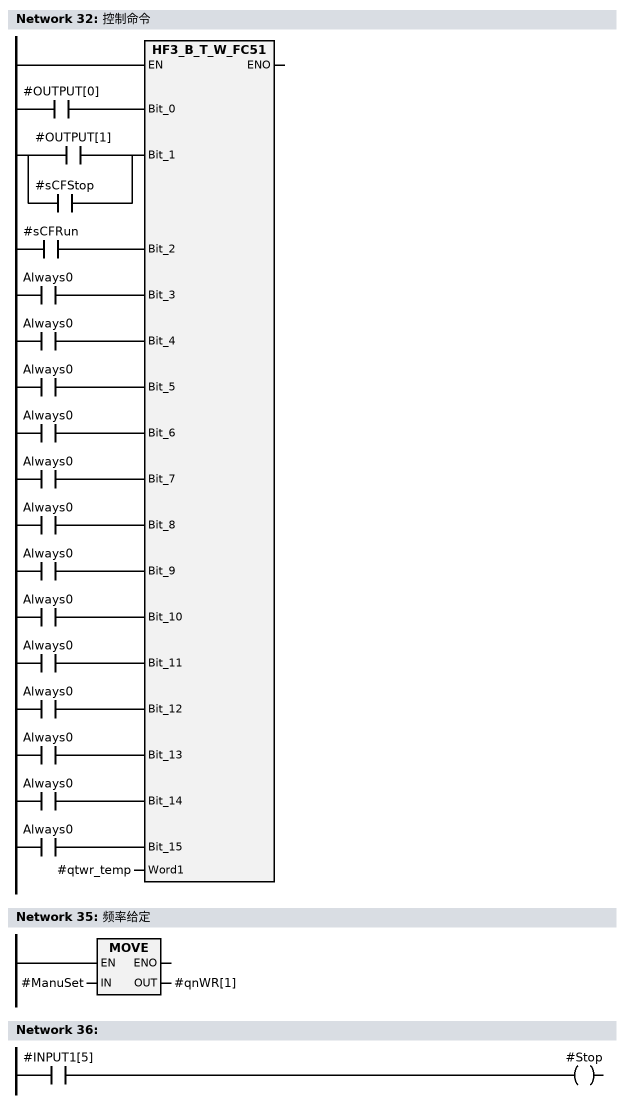
[picture p49: HF3_IMCC_TEF_FB2662 networks 32-36]
NETWORK
TITLE = 控制命令
      A     #OUTPUT[0];
      =     L 10.0;
      BLD   103;
      A(;
      O     #OUTPUT[1];
      O     #sCFStop;
      );
      =     L 10.1;
      BLD   103;
      A     #sCFRun;
      =     L 10.2;
      BLD   103;
      A     "Always0";
      =     L 10.3;
      BLD   103;
      A     "Always0";
      =     L 10.4;
      BLD   103;
      A     "Always0";
      =     L 10.5;
      BLD   103;
      A     "Always0";
      =     L 10.6;
      BLD   103;
      A     "Always0";
      =     L 10.7;
      BLD   103;
      A     "Always0";
      =     L 11.0;
      BLD   103;
      A     "Always0";
      =     L 11.1;
      BLD   103;
      A     "Always0";
      =     L 11.2;
      BLD   103;
      A     "Always0";
      =     L 11.3;
      BLD   103;
      A     "Always0";
      =     L 11.4;
      BLD   103;
      A     "Always0";
      =     L 11.5;
      BLD   103;
      A     "Always0";
      =     L 11.6;
      BLD   103;
      A     "Always0";
      =     L 11.7;
      BLD   103;
      CALL  "HF3_B_T_W_FC51" (
           Bit_0                    := L 10.0,
           Bit_1                    := L 10.1,
           Bit_2                    := L 10.2,
           Bit_3                    := L 10.3,
           Bit_4                    := L 10.4,
           Bit_5                    := L 10.5,
           Bit_6                    := L 10.6,
           Bit_7                    := L 10.7,
           Bit_8                    := L 11.0,
           Bit_9                    := L 11.1,
           Bit_10                   := L 11.2,
           Bit_11                   := L 11.3,
           Bit_12                   := L 11.4,
           Bit_13                   := L 11.5,
           Bit_14                   := L 11.6,
           Bit_15                   := L 11.7,
           Word1                    := #qtwr_temp);
      NOP   0;
NETWORK
TITLE = 参数传递
//控制命令输出
      CLR;
      L     #SCtrl;
      L     W#16#ABCD;
      <>I;
      JC    seiz;
      L     W#16#0;
      T     #qtwr_temp;
seiz: L     #qtwr_temp;
      T     #qnWR[0];
//tohmi输出
      L     #HMI_Adr;
      SLD   3;
      LAR1;
      OPN   DB [#DB_NO];
      L     #TOHMI_1;
      T     DBW [AR1,P#0.0];
      L     #TOHMI_2;
      T     DBW [AR1,P#2.0];
NETWORK
TITLE = 运行时间 故障次数
      A(;
      O     #INPUT1[3];
      O     #INPUT1[4];
      );
      =     L 10.0;
      BLD   103;
      A     #Flt;
      =     L 10.1;
      BLD   103;
      A     M 20.3;
      =     L 10.2;
      BLD   103;
      A     #SCtrl_Temp[12];
      =     L 10.4;
      BLD   103;
      A     #SCtrl_Temp[13];
      =     L 10.5;
      BLD   103;
      BLD   14;
      =     L 17.0;
      L     DINO;
      T     LW 15;
      CDB;
      OPN   DI [LW 15];
      TAR2  LD 11;
      A     L 10.0;
      =     DIX [AR2,P#136.0];
      A     L 10.1;
      =     DIX [AR2,P#136.1];
      A     L 10.2;
      =     DIX [AR2,P#136.2];
      A     L 10.4;
      =     DIX [AR2,P#136.4];
      A     L 10.5;
      =     DIX [AR2,P#136.5];
      +AR2  P#136.0;
      UC    "HF3_RunFaultSum";
      LAR2  LD 11;
      L     DID [AR2,P#138.0];
      T     DBD [AR2,P#58.0];
      L     DIW [AR2,P#142.0];
      T     DBW [AR2,P#64.0];
      L     DIW [AR2,P#144.0];
      T     DBW [AR2,P#62.0];
      CDB;
      BLD   15;
      NOP   0;
NETWORK
TITLE = 频率给定
      L     #ManuSet;
      T     #qnWR[1];
      NOP   0;
NETWORK
TITLE =
      A     #INPUT1[5];
      =     #Stop;
END_FUNCTION_BLOCK

FUNCTION_BLOCK "HF3_IMCC_KT_FB2671"	// FB 2671
VERSION : 0.1
VAR
  PT : TIME  := T#45S;
  KT_B1 : FB 2672;
END_VAR
BEGIN
NETWORK
TITLE =
// (network holds code this reader does not know; not shown)
END_FUNCTION_BLOCK

FUNCTION_BLOCK "HF3_IMCC_KT_FB2672"	// FB 2672
VERSION : 0.1
VAR_INPUT
  Main : BOOL ;	//1为大端 0为小端
  IN_RD : ARRAY  [0 .. 10 ] OF WORD ;
  HMI_Adr : INT ;
  SCtrl : WORD ;	//0单控1模控2启动3停止
  MCtrl : ARRAY  [0 .. 3 ] OF //模式控制
  BOOL ;
  Mode : ARRAY  [0 .. 15 ] OF //模式执行状态
  BOOL ;
  Open : BOOL ;	//风阀开连锁
  PT : TIME ;	//执行时间
  ALL : ARRAY  [0 .. 15 ] OF //单系统命令
  BOOL ;
  H_P_All_Ctrl : WORD ;	//全局命令
  FireAlarm : BOOL ;	//火灾报警
  BlockAlarm : BOOL ;	//阻塞报警
  ManuSet : INT ;	//手动频率给定
END_VAR
VAR_OUTPUT
  qnWR : ARRAY  [0 .. 1 ] OF WORD ;
  RT : REAL ;
  SumFlt : INT ;
  SumRun : INT ;
  refuse : BOOL ;
  Stop : BOOL ;	//风机控制
END_VAR
VAR
  IN_RD1 : WORD ;
  qtWR_1 : WORD ;
  TOHMI_1 : WORD ;
  TOHMI_2 : WORD ;
  qtwr_temp : WORD ;
  SFlag : BOOL ;	//单控标志
  McFlag : BOOL ;	//检修牌
  QTout : BOOL ;	//输出超时
  Flt : BOOL ;	//设备综合故障
  SingTout : BOOL ;	//单控超时
  Timeout : BOOL ;	//设备动作超时
  PID_EN : BOOL ;	//pid使能
  Fault : BOOL ;	//故障
  sCFRun : BOOL ;	//火灾启动
  sCFStop : BOOL ;	//火灾停止
  INPUT1 : ARRAY  [0 .. 15 ] OF //设备状态字
  BOOL ;
  OUTPUT : ARRAY  [0 .. 15 ] OF //输出状态字
  BOOL ;
  Ctrl : ARRAY  [0 .. 15 ] OF BOOL ;
  SCtrl_Temp : ARRAY  [0 .. 15 ] OF //HMI命令
  BOOL ;
  Latch : ARRAY  [0 .. 7 ] OF BOOL ;
  temp : ARRAY  [0 .. 1 ] OF BOOL ;
  h_P_all_temp : ARRAY  [0 .. 15 ] OF BOOL ;
  ton1 : SFB 4;
  ton2 : SFB 4;
  RunFaultSum : FB 2006;
END_VAR
VAR_TEMP
  AR2_Value : DWORD ;
  DI_NO : INT ;
  Data_Len : INT ;
  DB_NO : INT ;
END_VAR
BEGIN
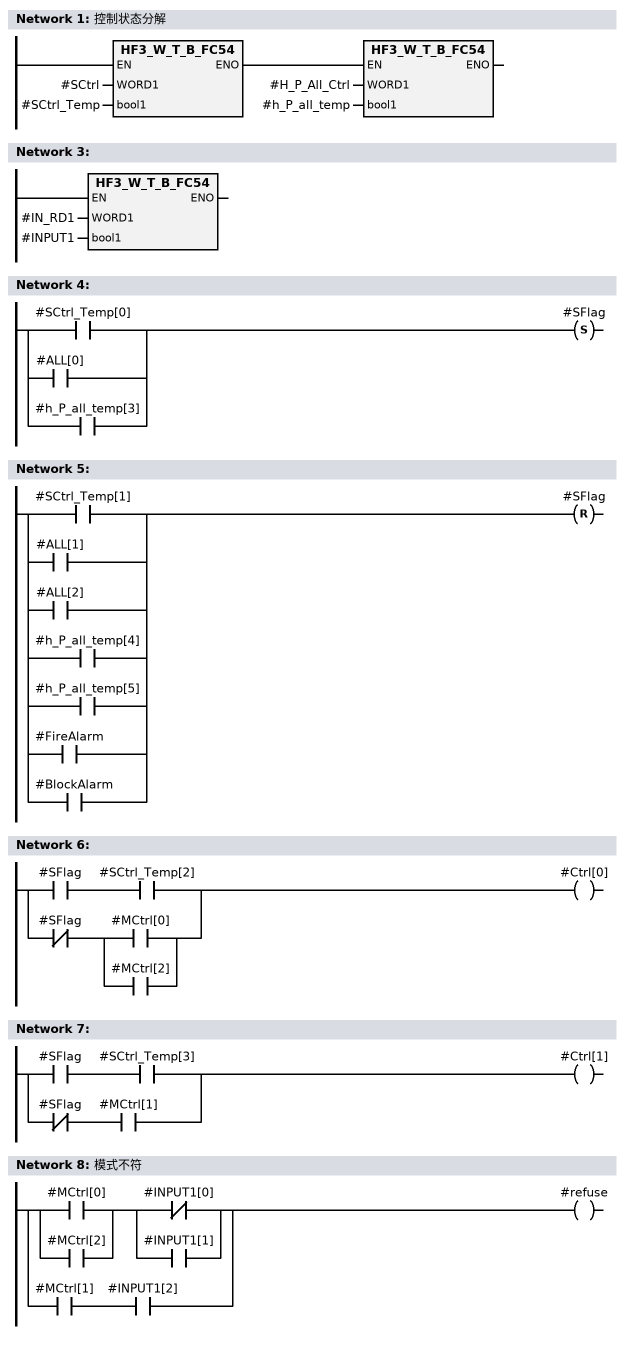
NETWORK
TITLE = 控制状态分解
      A(;
      CALL  "HF3_W_T_B_FC54" (
           WORD1                    := #SCtrl,
           bool1                    := #SCtrl_Temp);
      A     BR;
      );
      JNB   _001;
      CALL  "HF3_W_T_B_FC54" (
           WORD1                    := #H_P_All_Ctrl,
           bool1                    := #h_P_all_temp);
_001: NOP   0;
NETWORK
TITLE =
      TAR2;
      T     #AR2_Value;
      L     6002;
      T     #DB_NO;
      A     #Main;	//此端是否为大端
      JC    big;
      L     6004;
      T     #DB_NO;
big:  L     DINO;	//存储背景数据块号
      T     #DI_NO;
      OPN   DB [#DB_NO];	//打开
      L     #HMI_Adr;
      SLD   3;
      LAR1;
// *********************事故风机中DI状态读取**********************
      L     #IN_RD[0];	//第一个字中包含数字量信息
      T     #IN_RD1;
//初始化AR2寄存器用于AI量传递
      TAR2;
      AD    DW#16#FFFFFF;
      L     P##IN_RD;
      +D;
      OD    DW#16#85000000;
      LAR2;
//*********************事故风机中AI状态读取**********************
//读取模拟量输入
      L     13;
ilop: T     #Data_Len;
      L     W [AR2,P#2.0];	//智能低压点表新更新，第二个字开始为模拟量
      T     DBW [AR1,P#4.0];
      +AR1  P#2.0;
      +AR2  P#2.0;
      L     #Data_Len;
      LOOP  ilop;
//恢复AR2 DI寄存器
      L     #AR2_Value;
      LAR2;
//     OPN   DI [#DI_NO]
NETWORK
TITLE =
      CALL  "HF3_W_T_B_FC54" (
           WORD1                    := #IN_RD1,
           bool1                    := #INPUT1);
      NOP   0;
NETWORK
TITLE =
      O     #SCtrl_Temp[0];
      O     #ALL[0];
      O     #h_P_all_temp[3];
      S     #SFlag;
NETWORK
TITLE =
      O     #SCtrl_Temp[1];
      O     #ALL[1];
      O     #ALL[2];
      O     #h_P_all_temp[4];
      O     #h_P_all_temp[5];
      O     #FireAlarm;
      O     #BlockAlarm;
      R     #SFlag;
NETWORK
TITLE =
      A     #SFlag;
      A     #SCtrl_Temp[2];
      O;
      AN    #SFlag;
      A(;
      O     #MCtrl[0];
      O     #MCtrl[2];
      );
      =     #Ctrl[0];
NETWORK
TITLE =
      A     #SFlag;
      A     #SCtrl_Temp[3];
      O;
      AN    #SFlag;
      A     #MCtrl[1];
      =     #Ctrl[1];
NETWORK
TITLE = 模式不符
      A(;
      O     #MCtrl[0];
      O     #MCtrl[2];
      );
      A(;
      ON    #INPUT1[0];
      O     #INPUT1[1];
      );
      O;
      A     #MCtrl[1];
      A     #INPUT1[2];
      =     #refuse;
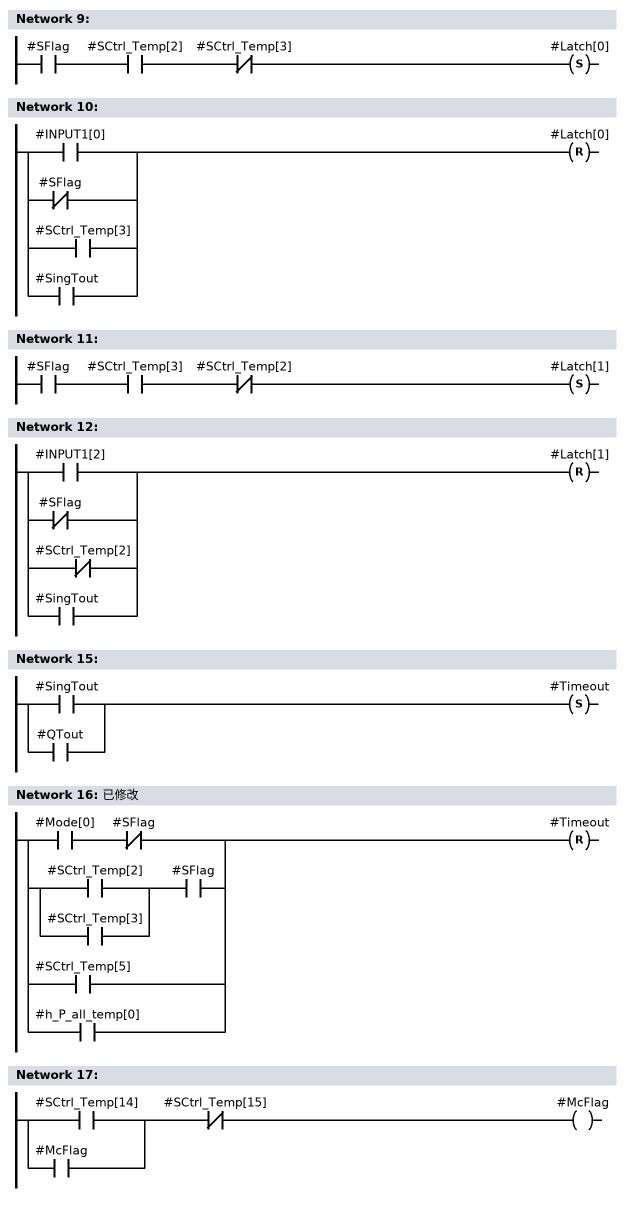
NETWORK
TITLE =
      A     #SFlag;
      A     #SCtrl_Temp[2];
      AN    #SCtrl_Temp[3];
      S     #Latch[0];
NETWORK
TITLE =
      O     #INPUT1[0];
      ON    #SFlag;
      O     #SCtrl_Temp[3];
      O     #SingTout;
      R     #Latch[0];
NETWORK
TITLE =
      A     #SFlag;
      A     #SCtrl_Temp[3];
      AN    #SCtrl_Temp[2];
      S     #Latch[1];
NETWORK
TITLE =
      O     #INPUT1[2];
      ON    #SFlag;
      ON    #SCtrl_Temp[2];
      O     #SingTout;
      R     #Latch[1];
NETWORK
TITLE =
      A(;
      O     #Latch[0];
      O     #Latch[1];
      );
      =     L 10.0;
      BLD   103;
      BLD   16;
      =     L 17.0;
      L     DINO;
      T     LW 15;
      CDB;
      OPN   DI [LW 15];
      TAR2  LD 11;
      A     L 10.0;
      =     DIX [AR2,P#86.0];
      L     DBD [AR2,P#34.0];
      T     DID [AR2,P#88.0];
      +AR2  P#86.0;
      UC    "TON";
      LAR2  LD 11;
      A     DIX [AR2,P#92.0];
      =     DBX [AR2,P#70.4];
      CDB;
      BLD   17;
      NOP   0;
NETWORK
TITLE =
      A(;
      O     #OUTPUT[0];
      O     #OUTPUT[1];
      );
      =     L 10.0;
      BLD   103;
      BLD   16;
      =     L 17.0;
      L     DINO;
      T     LW 15;
      CDB;
      OPN   DI [LW 15];
      TAR2  LD 11;
      A     L 10.0;
      =     DIX [AR2,P#108.0];
      L     DBD [AR2,P#34.0];
      T     DID [AR2,P#110.0];
      +AR2  P#108.0;
      UC    "TON";
      LAR2  LD 11;
      A     DIX [AR2,P#114.0];
      =     DBX [AR2,P#70.2];
      CDB;
      BLD   17;
      NOP   0;
NETWORK
TITLE =
      O     #SingTout;
      O     #QTout;
      S     #Timeout;
NETWORK
TITLE = 已修改
      A     #Mode[0];
      AN    #SFlag;
      O;
      A(;
      O     #SCtrl_Temp[2];
      O     #SCtrl_Temp[3];
      );
      A     #SFlag;
      O     #SCtrl_Temp[5];
      O     #h_P_all_temp[0];
      R     #Timeout;
NETWORK
TITLE =
      A(;
      O     #SCtrl_Temp[14];
      O     #McFlag;
      );
      AN    #SCtrl_Temp[15];
      =     #McFlag;
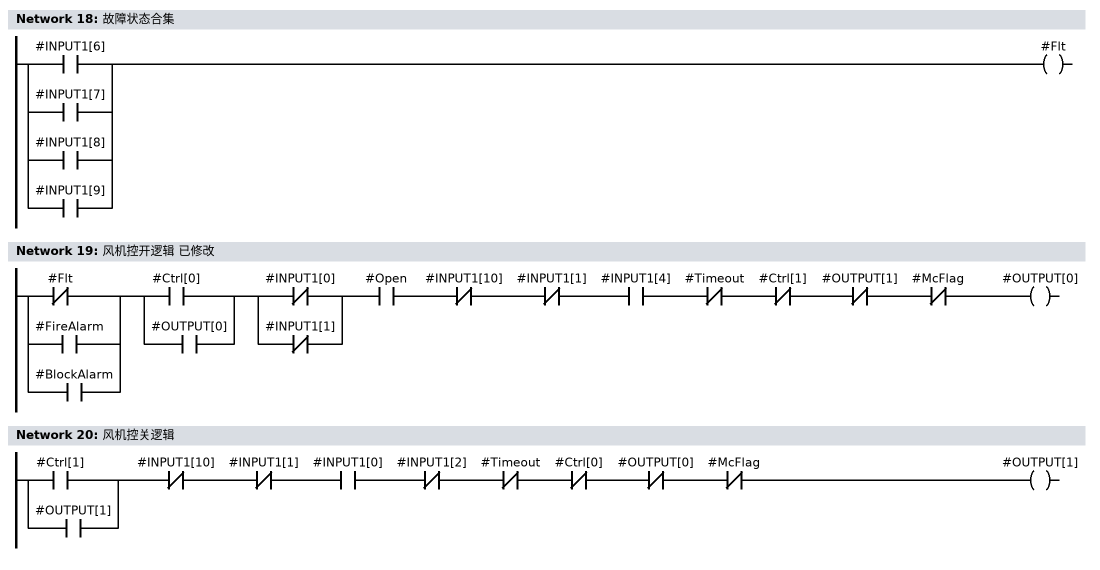
NETWORK
TITLE = 故障状态合集
      O     #INPUT1[6];
      O     #INPUT1[7];
      O     #INPUT1[8];
      O     #INPUT1[9];
      =     #Flt;
NETWORK
TITLE = 风机控开逻辑 已修改
      A(;
      ON    #Flt;
      O     #FireAlarm;
      O     #BlockAlarm;
      );
      A(;
      O     #Ctrl[0];
      O     #OUTPUT[0];
      );
      A(;
      ON    #INPUT1[0];
      ON    #INPUT1[1];
      );
      A     #Open;
      AN    #INPUT1[10];
      AN    #INPUT1[1];
      A     #INPUT1[4];
      AN    #Timeout;
      AN    #Ctrl[1];
      AN    #OUTPUT[1];
      AN    #McFlag;
      =     #OUTPUT[0];
NETWORK
TITLE = 风机控关逻辑
      A(;
      O     #Ctrl[1];
      O     #OUTPUT[1];
      );
      AN    #INPUT1[10];
      AN    #INPUT1[1];
      A     #INPUT1[0];
      AN    #INPUT1[2];
      AN    #Timeout;
      AN    #Ctrl[0];
      AN    #OUTPUT[0];
      AN    #McFlag;
      =     #OUTPUT[1];
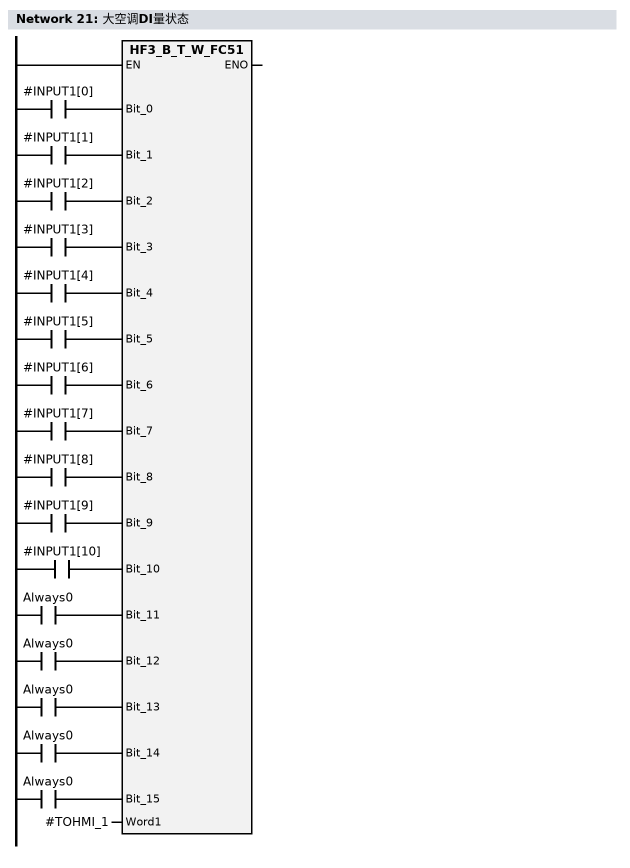
NETWORK
TITLE = 大空调DI量状态
      A     #INPUT1[0];
      =     L 10.0;
      BLD   103;
      A     #INPUT1[1];
      =     L 10.1;
      BLD   103;
      A     #INPUT1[2];
      =     L 10.2;
      BLD   103;
      A     #INPUT1[3];
      =     L 10.3;
      BLD   103;
      A     #INPUT1[4];
      =     L 10.4;
      BLD   103;
      A     #INPUT1[5];
      =     L 10.5;
      BLD   103;
      A     #INPUT1[6];
      =     L 10.6;
      BLD   103;
      A     #INPUT1[7];
      =     L 10.7;
      BLD   103;
      A     #INPUT1[8];
      =     L 11.0;
      BLD   103;
      A     #INPUT1[9];
      =     L 11.1;
      BLD   103;
      A     #INPUT1[10];
      =     L 11.2;
      BLD   103;
      A     "Always0";
      =     L 11.3;
      BLD   103;
      A     "Always0";
      =     L 11.4;
      BLD   103;
      A     "Always0";
      =     L 11.5;
      BLD   103;
      A     "Always0";
      =     L 11.6;
      BLD   103;
      A     "Always0";
      =     L 11.7;
      BLD   103;
      CALL  "HF3_B_T_W_FC51" (
           Bit_0                    := L 10.0,
           Bit_1                    := L 10.1,
           Bit_2                    := L 10.2,
           Bit_3                    := L 10.3,
           Bit_4                    := L 10.4,
           Bit_5                    := L 10.5,
           Bit_6                    := L 10.6,
           Bit_7                    := L 10.7,
           Bit_8                    := L 11.0,
           Bit_9                    := L 11.1,
           Bit_10                   := L 11.2,
           Bit_11                   := L 11.3,
           Bit_12                   := L 11.4,
           Bit_13                   := L 11.5,
           Bit_14                   := L 11.6,
           Bit_15                   := L 11.7,
           Word1                    := #TOHMI_1);
      NOP   0;
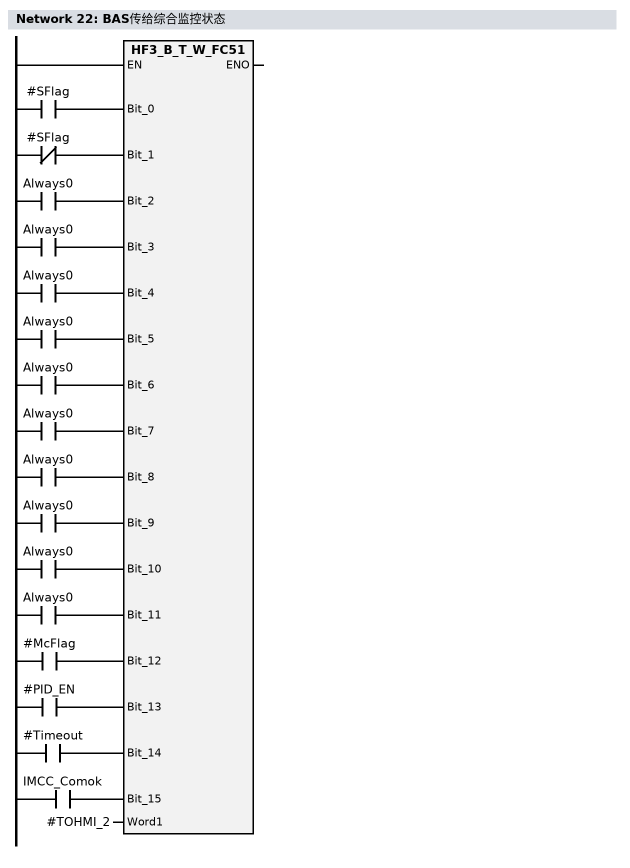
NETWORK
TITLE = BAS传给综合监控状态
//单模控、据动报警、检修牌、通讯状态
      A     #SFlag;
      =     L 10.0;
      BLD   103;
      AN    #SFlag;
      =     L 10.1;
      BLD   103;
      A     "Always0";
      =     L 10.2;
      BLD   103;
      A     "Always0";
      =     L 10.3;
      BLD   103;
      A     "Always0";
      =     L 10.4;
      BLD   103;
      A     "Always0";
      =     L 10.5;
      BLD   103;
      A     "Always0";
      =     L 10.6;
      BLD   103;
      A     "Always0";
      =     L 10.7;
      BLD   103;
      A     "Always0";
      =     L 11.0;
      BLD   103;
      A     "Always0";
      =     L 11.1;
      BLD   103;
      A     "Always0";
      =     L 11.2;
      BLD   103;
      A     "Always0";
      =     L 11.3;
      BLD   103;
      A     #McFlag;
      =     L 11.4;
      BLD   103;
      A     #PID_EN;
      =     L 11.5;
      BLD   103;
      A     #Timeout;
      =     L 11.6;
      BLD   103;
      A     "IMCC_Comok";
      =     L 11.7;
      BLD   103;
      CALL  "HF3_B_T_W_FC51" (
           Bit_0                    := L 10.0,
           Bit_1                    := L 10.1,
           Bit_2                    := L 10.2,
           Bit_3                    := L 10.3,
           Bit_4                    := L 10.4,
           Bit_5                    := L 10.5,
           Bit_6                    := L 10.6,
           Bit_7                    := L 10.7,
           Bit_8                    := L 11.0,
           Bit_9                    := L 11.1,
           Bit_10                   := L 11.2,
           Bit_11                   := L 11.3,
           Bit_12                   := L 11.4,
           Bit_13                   := L 11.5,
           Bit_14                   := L 11.6,
           Bit_15                   := L 11.7,
           Word1                    := #TOHMI_2);
      NOP   0;
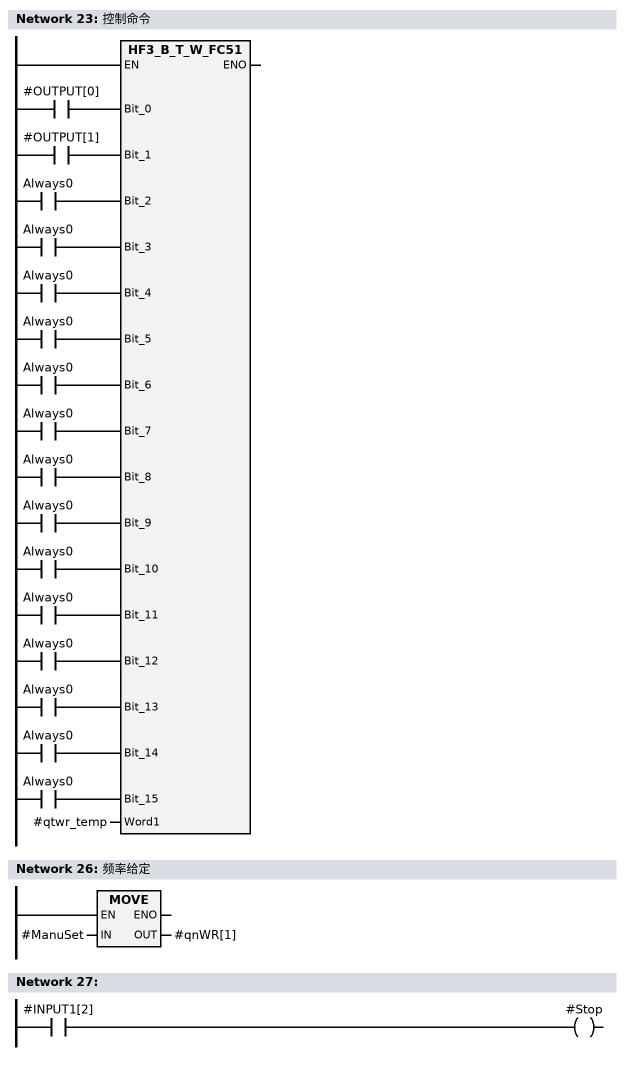
NETWORK
TITLE = 控制命令
      A     #OUTPUT[0];
      =     L 10.0;
      BLD   103;
      A     #OUTPUT[1];
      =     L 10.1;
      BLD   103;
      A     "Always0";
      =     L 10.2;
      BLD   103;
      A     "Always0";
      =     L 10.3;
      BLD   103;
      A     "Always0";
      =     L 10.4;
      BLD   103;
      A     "Always0";
      =     L 10.5;
      BLD   103;
      A     "Always0";
      =     L 10.6;
      BLD   103;
      A     "Always0";
      =     L 10.7;
      BLD   103;
      A     "Always0";
      =     L 11.0;
      BLD   103;
      A     "Always0";
      =     L 11.1;
      BLD   103;
      A     "Always0";
      =     L 11.2;
      BLD   103;
      A     "Always0";
      =     L 11.3;
      BLD   103;
      A     "Always0";
      =     L 11.4;
      BLD   103;
      A     "Always0";
      =     L 11.5;
      BLD   103;
      A     "Always0";
      =     L 11.6;
      BLD   103;
      A     "Always0";
      =     L 11.7;
      BLD   103;
      CALL  "HF3_B_T_W_FC51" (
           Bit_0                    := L 10.0,
           Bit_1                    := L 10.1,
           Bit_2                    := L 10.2,
           Bit_3                    := L 10.3,
           Bit_4                    := L 10.4,
           Bit_5                    := L 10.5,
           Bit_6                    := L 10.6,
           Bit_7                    := L 10.7,
           Bit_8                    := L 11.0,
           Bit_9                    := L 11.1,
           Bit_10                   := L 11.2,
           Bit_11                   := L 11.3,
           Bit_12                   := L 11.4,
           Bit_13                   := L 11.5,
           Bit_14                   := L 11.6,
           Bit_15                   := L 11.7,
           Word1                    := #qtwr_temp);
      NOP   0;
NETWORK
TITLE = 参数传递
//控制命令输出
      CLR;
      L     #SCtrl;
      L     W#16#ABCD;
      <>I;
      JC    seiz;
      L     W#16#0;
      T     #qtwr_temp;
seiz: L     #qtwr_temp;
      T     #qnWR[0];	//大空调开关控制字
//tohmi输出
      L     #HMI_Adr;
      SLD   3;
      LAR1;
      OPN   DB [#DB_NO];
      L     #TOHMI_1;
      T     DBW [AR1,P#0.0];
      L     #TOHMI_2;
      T     DBW [AR1,P#2.0];
NETWORK
TITLE =
      A(;
      O     #INPUT1[0];
      O     #INPUT1[1];
      );
      =     L 10.0;
      BLD   103;
      A     #Flt;
      =     L 10.1;
      BLD   103;
      A     M 20.5;
      =     L 10.2;
      BLD   103;
      A     #SCtrl_Temp[12];
      =     L 10.4;
      BLD   103;
      A     #SCtrl_Temp[13];
      =     L 10.5;
      BLD   103;
      BLD   14;
      =     L 17.0;
      L     DINO;
      T     LW 15;
      CDB;
      OPN   DI [LW 15];
      TAR2  LD 11;
      A     L 10.0;
      =     DIX [AR2,P#130.0];
      A     L 10.1;
      =     DIX [AR2,P#130.1];
      A     L 10.2;
      =     DIX [AR2,P#130.2];
      A     L 10.4;
      =     DIX [AR2,P#130.4];
      A     L 10.5;
      =     DIX [AR2,P#130.5];
      +AR2  P#130.0;
      UC    "HF3_RunFaultSum";
      LAR2  LD 11;
      L     DID [AR2,P#132.0];
      T     DBD [AR2,P#50.0];
      L     DIW [AR2,P#136.0];
      T     DBW [AR2,P#56.0];
      L     DIW [AR2,P#138.0];
      T     DBW [AR2,P#54.0];
      CDB;
      BLD   15;
      NOP   0;
NETWORK
TITLE = 频率给定
      L     #ManuSet;
      T     #qnWR[1];
      NOP   0;
NETWORK
TITLE =
      A     #INPUT1[2];
      =     #Stop;
END_FUNCTION_BLOCK

FUNCTION_BLOCK "HF3_IMCC_HPF_FB2681"	// FB 2681
VERSION : 0.1
VAR
  PT : TIME  := T#45S;
  HPF_A1 : FB 2682;
END_VAR
BEGIN
NETWORK
TITLE =
// (network holds code this reader does not know; not shown)
END_FUNCTION_BLOCK

FUNCTION_BLOCK "HF4_IMCC_HPF_FB2682"	// FB 2682
VERSION : 0.1
VAR_INPUT
  Main : BOOL ;
  IN_RD : ARRAY  [0 .. 7 ] OF WORD ;
  HMI_Adr : INT ;
  SCtrl : WORD ;	//01-单模23-启停
  MCtrl : ARRAY  [0 .. 3 ] OF //012-启动停止工频
  BOOL ;
  Mode : ARRAY  [0 .. 15 ] OF //012-开始结束时间表
  BOOL ;
  Open : BOOL ;	//连锁风阀开
  PT : TIME ;	//延迟时间
  ALL : ARRAY  [0 .. 15 ] OF //012-单控模控时间表
  BOOL ;
  H_P_All_Ctrl : WORD ;
  FireAlarm : BOOL ;	//火灾信号
  BlockAlarm : BOOL ;	//阻塞信号
  ManuSet : INT ;	//手动频率设定
END_VAR
VAR_OUTPUT
  qnWR : ARRAY  [0 .. 1 ] OF //0-频率1-启停
  WORD ;
  RT : REAL ;	//运行时间
  SumFlt : INT ;	//故障次数
  SumRun : INT ;	//运行次数
  Refuse : BOOL ;	//模式不符
  Stop : BOOL ;	//风机控制
END_VAR
VAR
  IN_RD1 : WORD ;
  qtWR : WORD ;
  TOHMI_1 : WORD ;
  TOHMI_2 : WORD ;
  qtwr_temp : WORD ;
  INPUT1 : ARRAY  [0 .. 15 ] OF BOOL ;
  OUTPUT : ARRAY  [0 .. 15 ] OF //01-启停
  BOOL ;
  Ctrl : ARRAY  [0 .. 15 ] OF //01-启停
  BOOL ;
  SCtrl_Temp : ARRAY  [0 .. 15 ] OF //01-单模23-启停
  BOOL ;
  H_P_All_Ctrl_Temp : ARRAY  [0 .. 15 ] OF BOOL ;
  Latch : ARRAY  [0 .. 7 ] OF //启停锁定
  BOOL ;
  McFlag : BOOL ;	//检修牌
  SFlag : BOOL ;	//单控标志
  SingTout : BOOL ;	//控制命令超时
  QTout : BOOL ;	//控制超时
  Timeout : BOOL ;	//超时
  Flt : BOOL ;	//设备综合故障
  PID_EN : BOOL ;	//PID使能
  Fault : BOOL ;
  TON1 : SFB 4;
  TON2 : SFB 4;
  RunFaultSum : FB 2006;
END_VAR
VAR_TEMP
  AR2_Value : DWORD ;
  DI_NO : INT ;
  Data_Len : INT ;
  DB_NO : INT ;
END_VAR
BEGIN
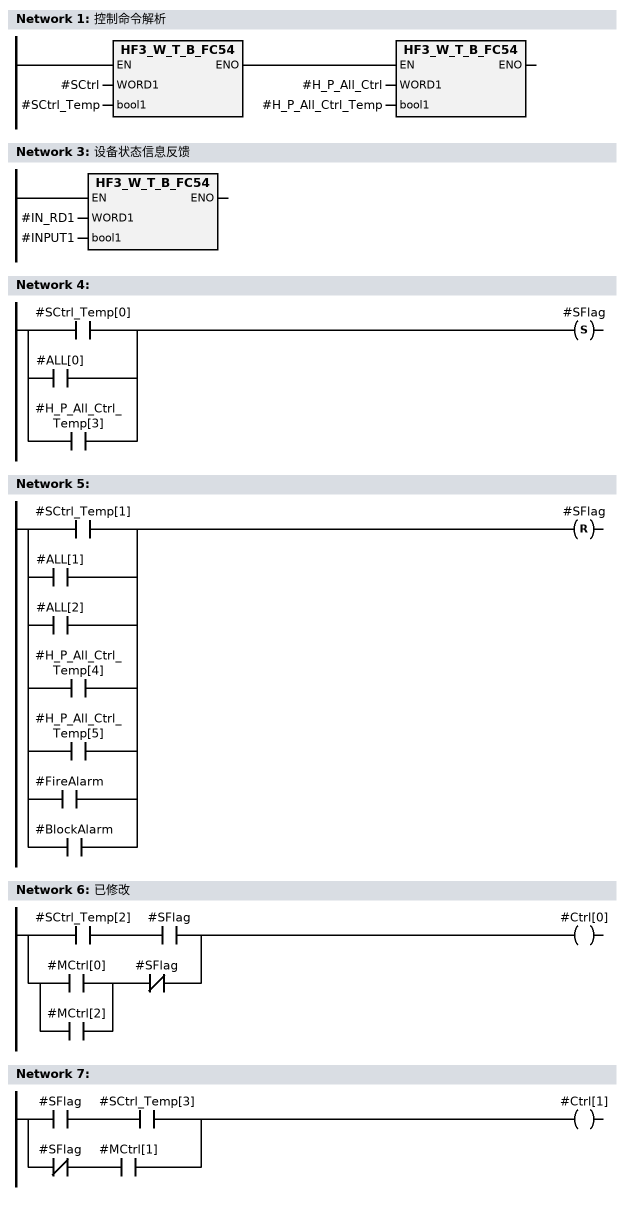
NETWORK
TITLE = 控制命令解析
      A(;
      CALL  "HF3_W_T_B_FC54" (
           WORD1                    := #SCtrl,
           bool1                    := #SCtrl_Temp);
      A     BR;
      );
      JNB   _001;
      CALL  "HF3_W_T_B_FC54" (
           WORD1                    := #H_P_All_Ctrl,
           bool1                    := #H_P_All_Ctrl_Temp);
_001: NOP   0;
NETWORK
TITLE = 状态信息读取
//第1个字BIT 0BAS
//第1个字BIT 1就地
//第1个字BIT 2变频/工频开关位置
//第1个字BIT 3变频运行状态
//第1个字BIT 4工频运行状态
//第1个字BIT 5变频器故障
//第1个字BIT 6变频器过载
//第1个字BIT 7电动机缺相
//
//
//第2个字频率反馈
//第3个字电动机电流A
//第4个字电动机电流B
//第5个字电动机电流C
//第6个字电动机电压A
//第7个字电动机电压B
//第8个字电动机电压C
//
      TAR2;
      T     #AR2_Value;
      L     6002;
      T     #DB_NO;
      A     #Main;	//此端是否为大端
      JC    big;
      L     6004;
      T     #DB_NO;
big:  L     DINO;	//存储背景数据块号
      T     #DI_NO;
      OPN   DB [#DB_NO];	//打开
      L     #HMI_Adr;
      SLD   3;
      LAR1;
// *********************事故风机中DI状态读取**********************
      L     #IN_RD[0];	//第一个字中包含数字量信息
      T     #IN_RD1;
//初始化AR2寄存器用于AI量传递
      TAR2;
      AD    DW#16#FFFFFF;
      L     P##IN_RD;
      +D;
      OD    DW#16#85000000;
      LAR2;
//*********************事故风机中AI状态读取**********************
//读取模拟量输入
      L     7;
ilop: T     #Data_Len;
      L     W [AR2,P#2.0];	//智能低压点表新更新，第二个字开始为模拟量
      T     DBW [AR1,P#4.0];
      +AR1  P#2.0;
      +AR2  P#2.0;
      L     #Data_Len;
      LOOP  ilop;
//恢复AR2 DI寄存器
      L     #AR2_Value;
      LAR2;
//     OPN   DI [#DI_NO]
NETWORK
TITLE = 设备状态信息反馈
      CALL  "HF3_W_T_B_FC54" (
           WORD1                    := #IN_RD1,
           bool1                    := #INPUT1);
      NOP   0;
NETWORK
TITLE =
      O     #SCtrl_Temp[0];
      O     #ALL[0];
      O     #H_P_All_Ctrl_Temp[3];
      S     #SFlag;
NETWORK
TITLE =
      O     #SCtrl_Temp[1];
      O     #ALL[1];
      O     #ALL[2];
      O     #H_P_All_Ctrl_Temp[4];
      O     #H_P_All_Ctrl_Temp[5];
      O     #FireAlarm;
      O     #BlockAlarm;
      R     #SFlag;
NETWORK
TITLE = 已修改
      A     #SCtrl_Temp[2];
      A     #SFlag;
      O;
      A(;
      O     #MCtrl[0];
      O     #MCtrl[2];
      );
      AN    #SFlag;
      =     #Ctrl[0];
NETWORK
TITLE =
      A     #SFlag;
      A     #SCtrl_Temp[3];
      O;
      AN    #SFlag;
      A     #MCtrl[1];
      =     #Ctrl[1];
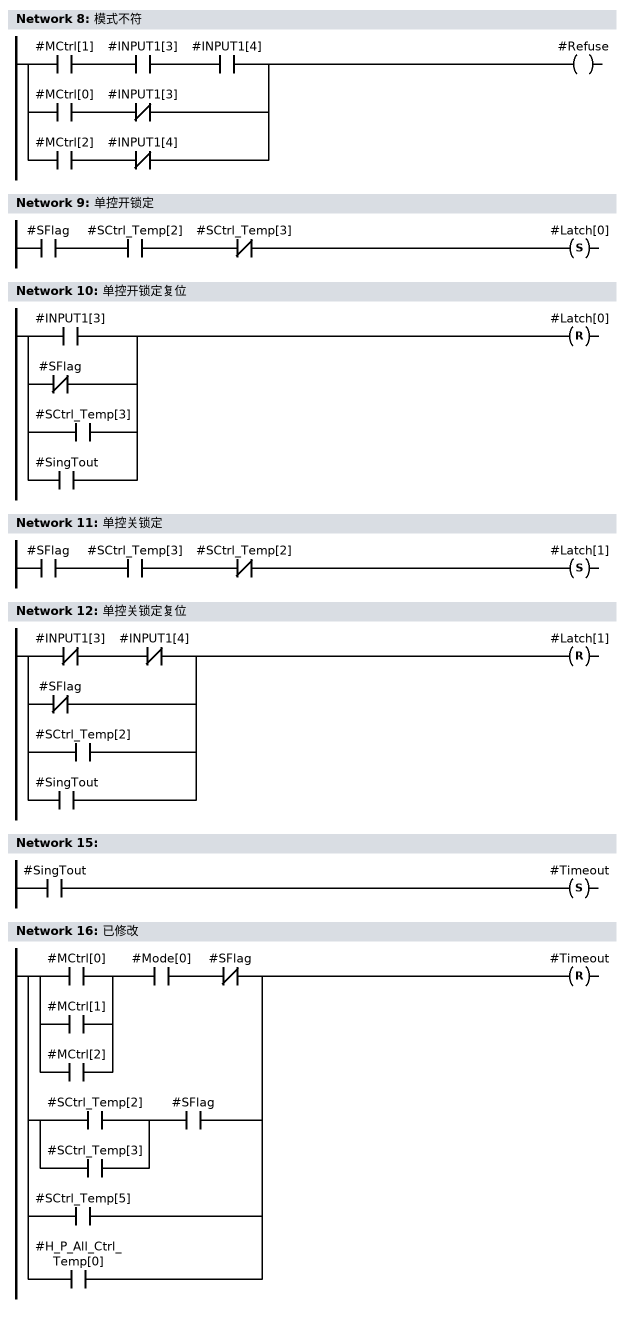
NETWORK
TITLE = 模式不符  
      A     #MCtrl[1];
      A     #INPUT1[3];
      A     #INPUT1[4];
      O;
      A     #MCtrl[0];
      AN    #INPUT1[3];
      O;
      A     #MCtrl[2];
      AN    #INPUT1[4];
      =     #Refuse;
NETWORK
TITLE = 单控开锁定
      A     #SFlag;
      A     #SCtrl_Temp[2];
      AN    #SCtrl_Temp[3];
      S     #Latch[0];
NETWORK
TITLE = 单控开锁定复位
      O     #INPUT1[3];
      ON    #SFlag;
      O     #SCtrl_Temp[3];
      O     #SingTout;
      R     #Latch[0];
NETWORK
TITLE = 单控关锁定
      A     #SFlag;
      A     #SCtrl_Temp[3];
      AN    #SCtrl_Temp[2];
      S     #Latch[1];
NETWORK
TITLE = 单控关锁定复位
      AN    #INPUT1[3];
      AN    #INPUT1[4];
      ON    #SFlag;
      O     #SCtrl_Temp[2];
      O     #SingTout;
      R     #Latch[1];
NETWORK
TITLE = 单控超时
      A(;
      O     #Latch[0];
      O     #Latch[1];
      );
      =     L 10.0;
      BLD   103;
      BLD   16;
      =     L 17.0;
      L     DINO;
      T     LW 15;
      CDB;
      OPN   DI [LW 15];
      TAR2  LD 11;
      A     L 10.0;
      =     DIX [AR2,P#78.0];
      L     DBD [AR2,P#28.0];
      T     DID [AR2,P#80.0];
      +AR2  P#78.0;
      UC    "TON";
      LAR2  LD 11;
      A     DIX [AR2,P#84.0];
      =     DBX [AR2,P#76.2];
      CDB;
      BLD   17;
      NOP   0;
NETWORK
TITLE = 控制命令超时
      A(;
      O     #OUTPUT[0];
      O     #OUTPUT[1];
      );
      =     L 10.0;
      BLD   103;
      BLD   16;
      =     L 17.0;
      L     DINO;
      T     LW 15;
      CDB;
      OPN   DI [LW 15];
      TAR2  LD 11;
      A     L 10.0;
      =     DIX [AR2,P#100.0];
      L     DBD [AR2,P#28.0];
      T     DID [AR2,P#102.0];
      +AR2  P#100.0;
      UC    "TON";
      LAR2  LD 11;
      A     DIX [AR2,P#106.0];
      =     DBX [AR2,P#76.3];
      CDB;
      BLD   17;
      NOP   0;
NETWORK
TITLE =
      A     #SingTout;
      S     #Timeout;
NETWORK
TITLE = 已修改
      A(;
      O     #MCtrl[0];
      O     #MCtrl[1];
      O     #MCtrl[2];
      );
      A     #Mode[0];
      AN    #SFlag;
      O;
      A(;
      O     #SCtrl_Temp[2];
      O     #SCtrl_Temp[3];
      );
      A     #SFlag;
      O     #SCtrl_Temp[5];
      O     #H_P_All_Ctrl_Temp[0];
      R     #Timeout;
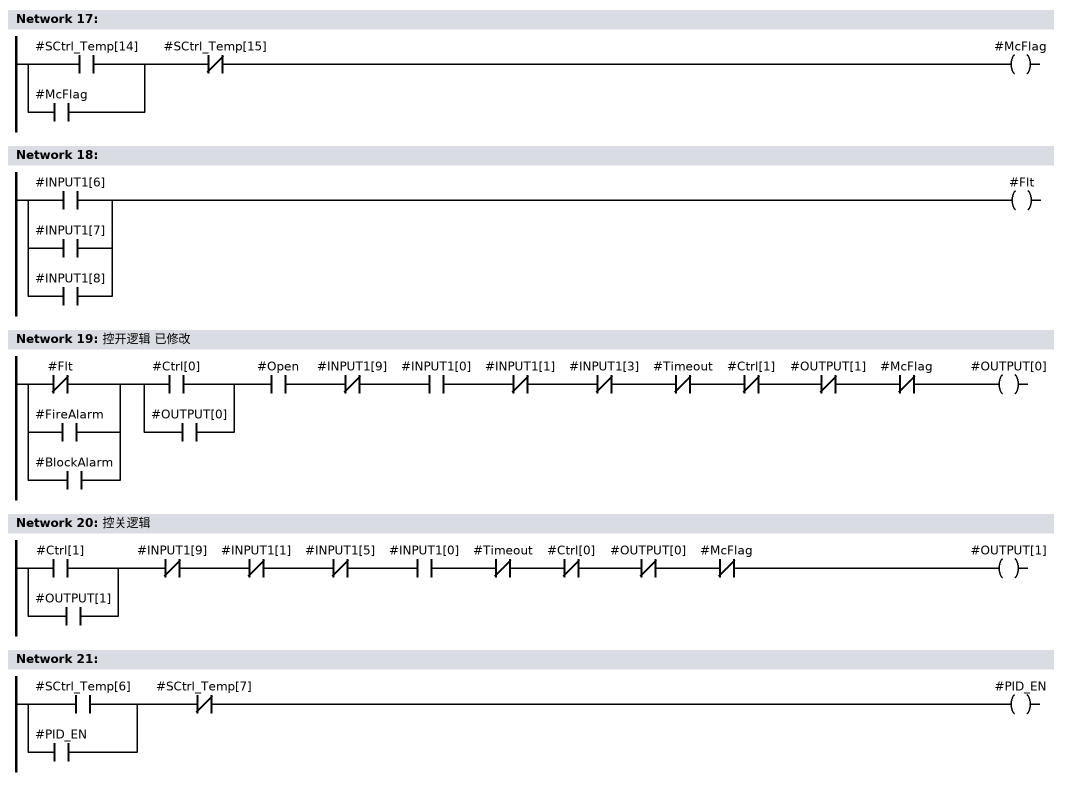
NETWORK
TITLE =
      A(;
      O     #SCtrl_Temp[14];
      O     #McFlag;
      );
      AN    #SCtrl_Temp[15];
      =     #McFlag;
NETWORK
TITLE =
      O     #INPUT1[6];
      O     #INPUT1[7];
      O     #INPUT1[8];
      =     #Flt;
NETWORK
TITLE = 控开逻辑 已修改
      A(;
      ON    #Flt;
      O     #FireAlarm;
      O     #BlockAlarm;
      );
      A(;
      O     #Ctrl[0];
      O     #OUTPUT[0];
      );
      A     #Open;
      AN    #INPUT1[9];
      A     #INPUT1[0];
      AN    #INPUT1[1];
      AN    #INPUT1[3];
      AN    #Timeout;
      AN    #Ctrl[1];
      AN    #OUTPUT[1];
      AN    #McFlag;
      =     #OUTPUT[0];
NETWORK
TITLE = 控关逻辑
      A(;
      O     #Ctrl[1];
      O     #OUTPUT[1];
      );
      AN    #INPUT1[9];
      AN    #INPUT1[1];
      AN    #INPUT1[5];
      A     #INPUT1[0];
      AN    #Timeout;
      AN    #Ctrl[0];
      AN    #OUTPUT[0];
      AN    #McFlag;
      =     #OUTPUT[1];
NETWORK
TITLE =
      A(;
      O     #SCtrl_Temp[6];
      O     #PID_EN;
      );
      AN    #SCtrl_Temp[7];
      =     #PID_EN;
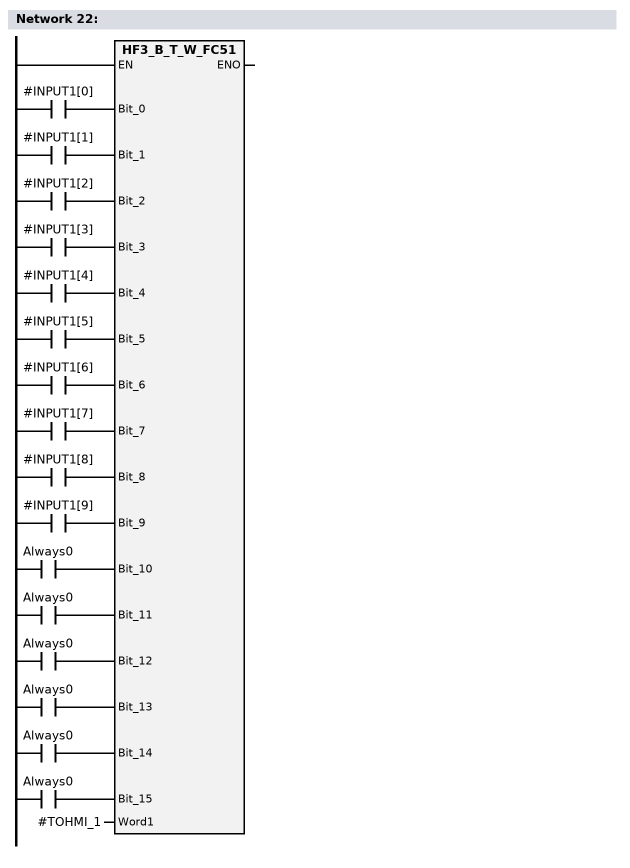
NETWORK
TITLE =
      A     #INPUT1[0];
      =     L 10.0;
      BLD   103;
      A     #INPUT1[1];
      =     L 10.1;
      BLD   103;
      A     #INPUT1[2];
      =     L 10.2;
      BLD   103;
      A     #INPUT1[3];
      =     L 10.3;
      BLD   103;
      A     #INPUT1[4];
      =     L 10.4;
      BLD   103;
      A     #INPUT1[5];
      =     L 10.5;
      BLD   103;
      A     #INPUT1[6];
      =     L 10.6;
      BLD   103;
      A     #INPUT1[7];
      =     L 10.7;
      BLD   103;
      A     #INPUT1[8];
      =     L 11.0;
      BLD   103;
      A     #INPUT1[9];
      =     L 11.1;
      BLD   103;
      A     "Always0";
      =     L 11.2;
      BLD   103;
      A     "Always0";
      =     L 11.3;
      BLD   103;
      A     "Always0";
      =     L 11.4;
      BLD   103;
      A     "Always0";
      =     L 11.5;
      BLD   103;
      A     "Always0";
      =     L 11.6;
      BLD   103;
      A     "Always0";
      =     L 11.7;
      BLD   103;
      CALL  "HF3_B_T_W_FC51" (
           Bit_0                    := L 10.0,
           Bit_1                    := L 10.1,
           Bit_2                    := L 10.2,
           Bit_3                    := L 10.3,
           Bit_4                    := L 10.4,
           Bit_5                    := L 10.5,
           Bit_6                    := L 10.6,
           Bit_7                    := L 10.7,
           Bit_8                    := L 11.0,
           Bit_9                    := L 11.1,
           Bit_10                   := L 11.2,
           Bit_11                   := L 11.3,
           Bit_12                   := L 11.4,
           Bit_13                   := L 11.5,
           Bit_14                   := L 11.6,
           Bit_15                   := L 11.7,
           Word1                    := #TOHMI_1);
      NOP   0;
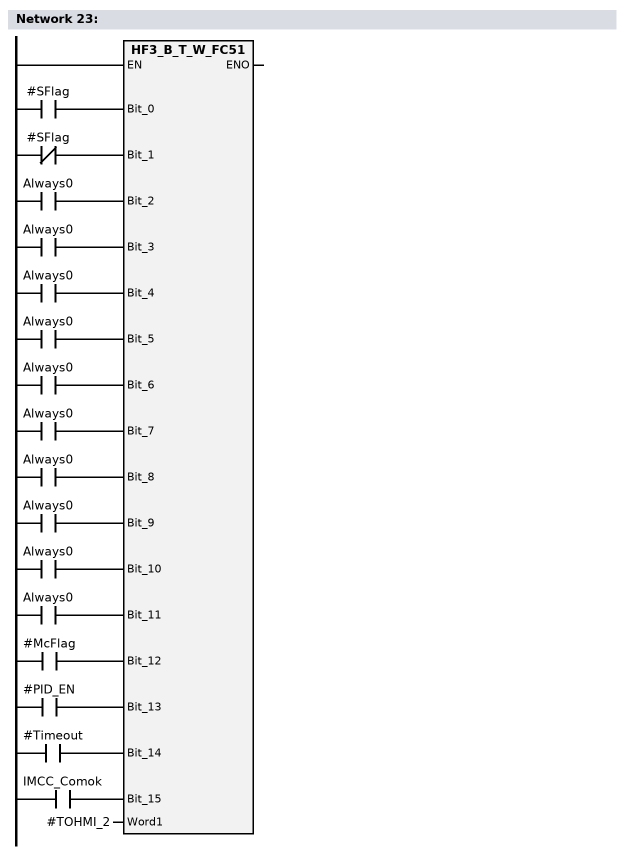
NETWORK
TITLE =
      A     #SFlag;
      =     L 10.0;
      BLD   103;
      AN    #SFlag;
      =     L 10.1;
      BLD   103;
      A     "Always0";
      =     L 10.2;
      BLD   103;
      A     "Always0";
      =     L 10.3;
      BLD   103;
      A     "Always0";
      =     L 10.4;
      BLD   103;
      A     "Always0";
      =     L 10.5;
      BLD   103;
      A     "Always0";
      =     L 10.6;
      BLD   103;
      A     "Always0";
      =     L 10.7;
      BLD   103;
      A     "Always0";
      =     L 11.0;
      BLD   103;
      A     "Always0";
      =     L 11.1;
      BLD   103;
      A     "Always0";
      =     L 11.2;
      BLD   103;
      A     "Always0";
      =     L 11.3;
      BLD   103;
      A     #McFlag;
      =     L 11.4;
      BLD   103;
      A     #PID_EN;
      =     L 11.5;
      BLD   103;
      A     #Timeout;
      =     L 11.6;
      BLD   103;
      A     "IMCC_Comok";
      =     L 11.7;
      BLD   103;
      CALL  "HF3_B_T_W_FC51" (
           Bit_0                    := L 10.0,
           Bit_1                    := L 10.1,
           Bit_2                    := L 10.2,
           Bit_3                    := L 10.3,
           Bit_4                    := L 10.4,
           Bit_5                    := L 10.5,
           Bit_6                    := L 10.6,
           Bit_7                    := L 10.7,
           Bit_8                    := L 11.0,
           Bit_9                    := L 11.1,
           Bit_10                   := L 11.2,
           Bit_11                   := L 11.3,
           Bit_12                   := L 11.4,
           Bit_13                   := L 11.5,
           Bit_14                   := L 11.6,
           Bit_15                   := L 11.7,
           Word1                    := #TOHMI_2);
      NOP   0;
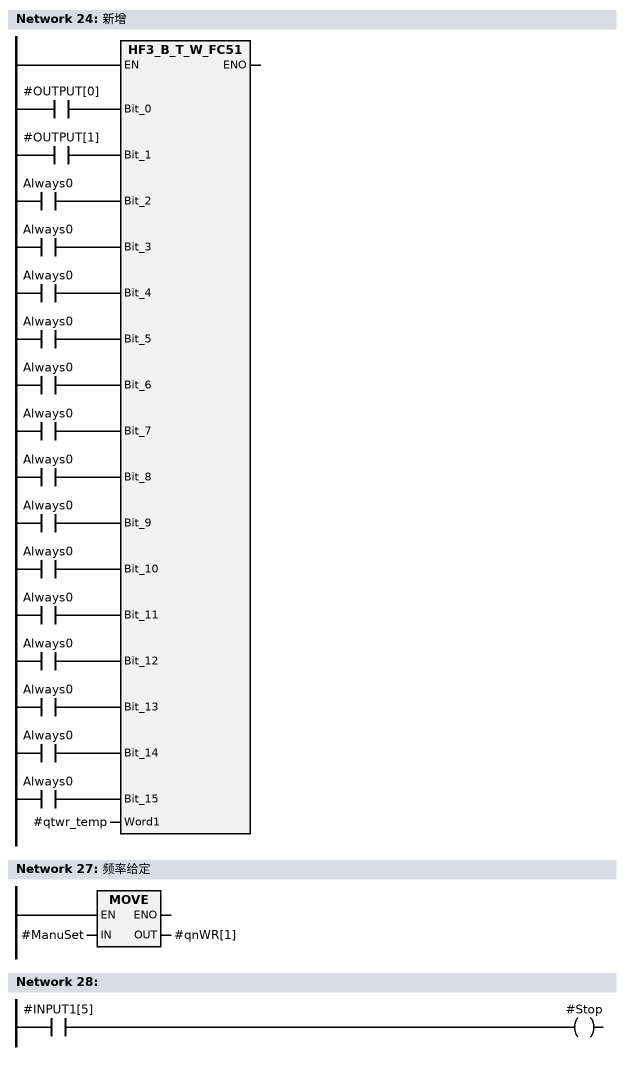
NETWORK
TITLE = 新增
      A     #OUTPUT[0];
      =     L 10.0;
      BLD   103;
      A     #OUTPUT[1];
      =     L 10.1;
      BLD   103;
      A     "Always0";
      =     L 10.2;
      BLD   103;
      A     "Always0";
      =     L 10.3;
      BLD   103;
      A     "Always0";
      =     L 10.4;
      BLD   103;
      A     "Always0";
      =     L 10.5;
      BLD   103;
      A     "Always0";
      =     L 10.6;
      BLD   103;
      A     "Always0";
      =     L 10.7;
      BLD   103;
      A     "Always0";
      =     L 11.0;
      BLD   103;
      A     "Always0";
      =     L 11.1;
      BLD   103;
      A     "Always0";
      =     L 11.2;
      BLD   103;
      A     "Always0";
      =     L 11.3;
      BLD   103;
      A     "Always0";
      =     L 11.4;
      BLD   103;
      A     "Always0";
      =     L 11.5;
      BLD   103;
      A     "Always0";
      =     L 11.6;
      BLD   103;
      A     "Always0";
      =     L 11.7;
      BLD   103;
      CALL  "HF3_B_T_W_FC51" (
           Bit_0                    := L 10.0,
           Bit_1                    := L 10.1,
           Bit_2                    := L 10.2,
           Bit_3                    := L 10.3,
           Bit_4                    := L 10.4,
           Bit_5                    := L 10.5,
           Bit_6                    := L 10.6,
           Bit_7                    := L 10.7,
           Bit_8                    := L 11.0,
           Bit_9                    := L 11.1,
           Bit_10                   := L 11.2,
           Bit_11                   := L 11.3,
           Bit_12                   := L 11.4,
           Bit_13                   := L 11.5,
           Bit_14                   := L 11.6,
           Bit_15                   := L 11.7,
           Word1                    := #qtwr_temp);
      NOP   0;
NETWORK
TITLE =
//控制命令输出
      CLR;
      L     #SCtrl;
      L     W#16#ABCD;
      <>I;
      JC    seiz;
      L     W#16#0;
      T     #qtwr_temp;
seiz: L     #qtwr_temp;
      T     #qnWR[0];
//tohmi输出
      L     #HMI_Adr;
      SLD   3;
      LAR1;
      OPN   DB [#DB_NO];
      L     #TOHMI_1;
      T     DBW [AR1,P#0.0];
      L     #TOHMI_2;
      T     DBW [AR1,P#2.0];
NETWORK
TITLE =
      A(;
      O     #INPUT1[3];
      O     #INPUT1[4];
      );
      =     L 10.0;
      BLD   103;
      A     #Flt;
      =     L 10.1;
      BLD   103;
      A     M 20.3;
      =     L 10.2;
      BLD   103;
      A     #SCtrl_Temp[12];
      =     L 10.4;
      BLD   103;
      A     #SCtrl_Temp[13];
      =     L 10.5;
      BLD   103;
      BLD   14;
      =     L 17.0;
      L     DINO;
      T     LW 15;
      CDB;
      OPN   DI [LW 15];
      TAR2  LD 11;
      A     L 10.0;
      =     DIX [AR2,P#122.0];
      A     L 10.1;
      =     DIX [AR2,P#122.1];
      A     L 10.2;
      =     DIX [AR2,P#122.2];
      A     L 10.4;
      =     DIX [AR2,P#122.4];
      A     L 10.5;
      =     DIX [AR2,P#122.5];
      +AR2  P#122.0;
      UC    "HF3_RunFaultSum";
      LAR2  LD 11;
      L     DID [AR2,P#124.0];
      T     DBD [AR2,P#44.0];
      L     DIW [AR2,P#128.0];
      T     DBW [AR2,P#50.0];
      L     DIW [AR2,P#130.0];
      T     DBW [AR2,P#48.0];
      CDB;
      BLD   15;
      NOP   0;
NETWORK
TITLE = 频率给定
      L     #ManuSet;
      T     #qnWR[1];
      NOP   0;
NETWORK
TITLE =
      A     #INPUT1[5];
      =     #Stop;
END_FUNCTION_BLOCK

FUNCTION_BLOCK "HF3_IMCC_FJ_FB2691"	// FB 2691
TITLE = IMCC系统风机
//智能低压系统A端所有小风机
//
VERSION : 0.1
VAR
  PT : TIME  := T#45S;
  T1_XSF_B2 : FB 2692;
  T1_XPY_B2 : FB 2692;
  RFP_B1 : FB 2692;
  K1_HPF_B1 : FB 2692;
  K2_HPF_B1 : FB 2692;
  K3_HPF_B1 : FB 2692;
  T1_XPF_B1 : FB 2692;
  T4_XPF_B1 : FB 2692;
  K2_XK_B1 : FB 2692;
  K3_XK_B1 : FB 2692;
  K2_XK_B2 : FB 2692;
  K3_XK_B3 : FB 2692;
  T1_XSF_B1 : FB 2692;
  T5_XPF_B1 : FB 2692;
  K4_XK_A1 : FB 2692;
  K4_HPF_A1 : FB 2692;
  T6_XSF_A1 : FB 2692;
  T6_XPF_A1 : FB 2692;
  T7_XPF_A1 : FB 2692;
END_VAR
BEGIN
NETWORK
TITLE = K4_XK_A1
      A     "Always0";
      =     L 0.0;
      BLD   103;
      A(;
      O     "IMCC_LOCK".K4_DT_A1_Open;
      O     "IMCC_LOCK".K4_DT_A3_Open;
      );
      =     L 0.1;
      BLD   103;
      A     "Maste_To_Slave_Mod_DB".FireAlarm;
      =     L 0.2;
      BLD   103;
      A     "Maste_To_Slave_Mod_DB".BlockAlarm;
      =     L 0.3;
      BLD   103;
      BLD   14;
      =     L 7.0;
      L     DINO;
      T     LW 5;
      CDB;
      OPN   DI [LW 5];
      TAR2  LD 1;
      A     L 0.0;
      =     DIX [AR2,P#1768.0];
      BLD   11;
      L     W#16#1002;
      T     LW 10;
      L     8;
      T     LW 12;
      L     2291;
      T     LW 14;
      L     P#DBX 68.0;
      T     LD 16;
      L     W#16#1002;
      T     LW 20;
      L     8;
      T     LW 22;
      L     DINO;
      T     LW 24;
      +AR2  P#1770.0;
      TAR2;
      LAR2  LD 1;
      T     LD 26;
      UC    "BLKMOV";
      {     P#L 10.0, P#L 8.0, P#L 20.0 };
      L     608;
      T     DIW [AR2,P#1778.0];
      OPN   DI 6040;
      L     DIW 148;
      OPN   DI [LW 5];
      T     DIW [AR2,P#1780.0];
      BLD   11;
      L     W#16#1002;
      T     LW 10;
      L     2;
      T     LW 12;
      L     7004;
      T     LW 14;
      L     P#DBX 54.0;
      T     LD 16;
      L     W#16#1002;
      T     LW 20;
      L     2;
      T     LW 22;
      L     DINO;
      T     LW 24;
      +AR2  P#1782.0;
      TAR2;
      LAR2  LD 1;
      T     LD 26;
      UC    "BLKMOV";
      {     P#L 10.0, P#L 8.0, P#L 20.0 };
      BLD   11;
      L     W#16#1002;
      T     LW 10;
      L     2;
      T     LW 12;
      L     7005;
      T     LW 14;
      L     P#DBX 4.0;
      T     LD 16;
      L     W#16#1002;
      T     LW 20;
      L     2;
      T     LW 22;
      L     DINO;
      T     LW 24;
      +AR2  P#1784.0;
      TAR2;
      LAR2  LD 1;
      T     LD 26;
      UC    "BLKMOV";
      {     P#L 10.0, P#L 8.0, P#L 20.0 };
      A     L 0.1;
      =     DIX [AR2,P#1786.0];
      L     DBD [AR2,P#0.0];
      T     DID [AR2,P#1788.0];
      BLD   11;
      L     W#16#1002;
      T     LW 10;
      L     2;
      T     LW 12;
      L     7005;
      T     LW 14;
      L     P#DBX 34.0;
      T     LD 16;
      L     W#16#1002;
      T     LW 20;
      L     2;
      T     LW 22;
      L     DINO;
      T     LW 24;
      +AR2  P#1792.0;
      TAR2;
      LAR2  LD 1;
      T     LD 26;
      UC    "BLKMOV";
      {     P#L 10.0, P#L 8.0, P#L 20.0 };
      OPN   DI 7005;
      L     DIW 312;
      OPN   DI [LW 5];
      T     DIW [AR2,P#1794.0];
      A     L 0.2;
      =     DIX [AR2,P#1796.0];
      A     L 0.3;
      =     DIX [AR2,P#1796.1];
      +AR2  P#1768.0;
      UC    "HF3_IMCC_FJ_FB2692";
      LAR2  LD 1;
      L     DIW [AR2,P#1798.0];
      OPN   DI 2292;
      T     DIW 20;
      OPN   DI [LW 5];
      L     DID [AR2,P#1800.0];
      OPN   DI 6004;
      T     DID 616;
      OPN   DI [LW 5];
      L     DIW [AR2,P#1804.0];
      OPN   DI 6004;
      T     DIW 620;
      OPN   DI [LW 5];
      A     DIX [AR2,P#1808.0];
      OPN   DI 7006;
      =     DIX 4.6;
      OPN   DI [LW 5];
      A     DIX [AR2,P#1808.1];
      OPN   DI 2555;
      =     DIX 2.7;
      OPN   DI [LW 5];
      CDB;
      BLD   15;
      NOP   0;
NETWORK
TITLE = K4_HPF_A1
      A     "Always0";
      =     L 0.0;
      BLD   103;
      A(;
      O     "IMCC_LOCK".K4_DT_A2_Open;
      O     "IMCC_LOCK".K4_DT_A3_Open;
      );
      =     L 0.1;
      BLD   103;
      A     "Maste_To_Slave_Mod_DB".FireAlarm;
      =     L 0.2;
      BLD   103;
      A     "Maste_To_Slave_Mod_DB".BlockAlarm;
      =     L 0.3;
      BLD   103;
      BLD   14;
      =     L 7.0;
      L     DINO;
      T     LW 5;
      CDB;
      OPN   DI [LW 5];
      TAR2  LD 1;
      A     L 0.0;
      =     DIX [AR2,P#1894.0];
      BLD   11;
      L     W#16#1002;
      T     LW 10;
      L     8;
      T     LW 12;
      L     2291;
      T     LW 14;
      L     P#DBX 36.0;
      T     LD 16;
      L     W#16#1002;
      T     LW 20;
      L     8;
      T     LW 22;
      L     DINO;
      T     LW 24;
      +AR2  P#1896.0;
      TAR2;
      LAR2  LD 1;
      T     LD 26;
      UC    "BLKMOV";
      {     P#L 10.0, P#L 8.0, P#L 20.0 };
      L     622;
      T     DIW [AR2,P#1904.0];
      OPN   DI 6040;
      L     DIW 150;
      OPN   DI [LW 5];
      T     DIW [AR2,P#1906.0];
      BLD   11;
      L     W#16#1002;
      T     LW 10;
      L     2;
      T     LW 12;
      L     7004;
      T     LW 14;
      L     P#DBX 56.0;
      T     LD 16;
      L     W#16#1002;
      T     LW 20;
      L     2;
      T     LW 22;
      L     DINO;
      T     LW 24;
      +AR2  P#1908.0;
      TAR2;
      LAR2  LD 1;
      T     LD 26;
      UC    "BLKMOV";
      {     P#L 10.0, P#L 8.0, P#L 20.0 };
      BLD   11;
      L     W#16#1002;
      T     LW 10;
      L     2;
      T     LW 12;
      L     7005;
      T     LW 14;
      L     P#DBX 4.0;
      T     LD 16;
      L     W#16#1002;
      T     LW 20;
      L     2;
      T     LW 22;
      L     DINO;
      T     LW 24;
      +AR2  P#1910.0;
      TAR2;
      LAR2  LD 1;
      T     LD 26;
      UC    "BLKMOV";
      {     P#L 10.0, P#L 8.0, P#L 20.0 };
      A     L 0.1;
      =     DIX [AR2,P#1912.0];
      L     DBD [AR2,P#0.0];
      T     DID [AR2,P#1914.0];
      BLD   11;
      L     W#16#1002;
      T     LW 10;
      L     2;
      T     LW 12;
      L     7005;
      T     LW 14;
      L     P#DBX 34.0;
      T     LD 16;
      L     W#16#1002;
      T     LW 20;
      L     2;
      T     LW 22;
      L     DINO;
      T     LW 24;
      +AR2  P#1918.0;
      TAR2;
      LAR2  LD 1;
      T     LD 26;
      UC    "BLKMOV";
      {     P#L 10.0, P#L 8.0, P#L 20.0 };
      OPN   DI 7005;
      L     DIW 312;
      OPN   DI [LW 5];
      T     DIW [AR2,P#1920.0];
      A     L 0.2;
      =     DIX [AR2,P#1922.0];
      A     L 0.3;
      =     DIX [AR2,P#1922.1];
      +AR2  P#1894.0;
      UC    "HF3_IMCC_FJ_FB2692";
      LAR2  LD 1;
      L     DIW [AR2,P#1924.0];
      OPN   DI 2292;
      T     DIW 12;
      OPN   DI [LW 5];
      L     DID [AR2,P#1926.0];
      OPN   DI 6004;
      T     DID 630;
      OPN   DI [LW 5];
      L     DIW [AR2,P#1930.0];
      OPN   DI 6004;
      T     DIW 634;
      OPN   DI [LW 5];
      A     DIX [AR2,P#1934.0];
      OPN   DI 7006;
      =     DIX 4.7;
      OPN   DI [LW 5];
      A     DIX [AR2,P#1934.1];
      OPN   DI 2555;
      =     DIX 3.0;
      OPN   DI [LW 5];
      CDB;
      BLD   15;
      NOP   0;
NETWORK
TITLE = T6_SXF_A1
      A     "Always0";
      =     L 0.0;
      BLD   103;
      A     "IMCC_LOCK".T6_D_A1_Open;
      =     L 0.1;
      BLD   103;
      A     "Maste_To_Slave_Mod_DB".FireAlarm;
      =     L 0.2;
      BLD   103;
      A     "Maste_To_Slave_Mod_DB".BlockAlarm;
      =     L 0.3;
      BLD   103;
      BLD   14;
      =     L 7.0;
      L     DINO;
      T     LW 5;
      CDB;
      OPN   DI [LW 5];
      TAR2  LD 1;
      A     L 0.0;
      =     DIX [AR2,P#2020.0];
      BLD   11;
      L     W#16#1002;
      T     LW 10;
      L     8;
      T     LW 12;
      L     2291;
      T     LW 14;
      L     P#DBX 12.0;
      T     LD 16;
      L     W#16#1002;
      T     LW 20;
      L     8;
      T     LW 22;
      L     DINO;
      T     LW 24;
      +AR2  P#2022.0;
      TAR2;
      LAR2  LD 1;
      T     LD 26;
      UC    "BLKMOV";
      {     P#L 10.0, P#L 8.0, P#L 20.0 };
      L     552;
      T     DIW [AR2,P#2030.0];
      OPN   DI 6040;
      L     DIW 228;
      OPN   DI [LW 5];
      T     DIW [AR2,P#2032.0];
      BLD   11;
      L     W#16#1002;
      T     LW 10;
      L     2;
      T     LW 12;
      L     7004;
      T     LW 14;
      L     P#DBX 66.0;
      T     LD 16;
      L     W#16#1002;
      T     LW 20;
      L     2;
      T     LW 22;
      L     DINO;
      T     LW 24;
      +AR2  P#2034.0;
      TAR2;
      LAR2  LD 1;
      T     LD 26;
      UC    "BLKMOV";
      {     P#L 10.0, P#L 8.0, P#L 20.0 };
      BLD   11;
      L     W#16#1002;
      T     LW 10;
      L     2;
      T     LW 12;
      L     7005;
      T     LW 14;
      L     P#DBX 6.0;
      T     LD 16;
      L     W#16#1002;
      T     LW 20;
      L     2;
      T     LW 22;
      L     DINO;
      T     LW 24;
      +AR2  P#2036.0;
      TAR2;
      LAR2  LD 1;
      T     LD 26;
      UC    "BLKMOV";
      {     P#L 10.0, P#L 8.0, P#L 20.0 };
      A     L 0.1;
      =     DIX [AR2,P#2038.0];
      L     DBD [AR2,P#0.0];
      T     DID [AR2,P#2040.0];
      BLD   11;
      L     W#16#1002;
      T     LW 10;
      L     2;
      T     LW 12;
      L     7005;
      T     LW 14;
      L     P#DBX 36.0;
      T     LD 16;
      L     W#16#1002;
      T     LW 20;
      L     2;
      T     LW 22;
      L     DINO;
      T     LW 24;
      +AR2  P#2044.0;
      TAR2;
      LAR2  LD 1;
      T     LD 26;
      UC    "BLKMOV";
      {     P#L 10.0, P#L 8.0, P#L 20.0 };
      OPN   DI 7005;
      L     DIW 312;
      OPN   DI [LW 5];
      T     DIW [AR2,P#2046.0];
      A     L 0.2;
      =     DIX [AR2,P#2048.0];
      A     L 0.3;
      =     DIX [AR2,P#2048.1];
      +AR2  P#2020.0;
      UC    "HF3_IMCC_FJ_FB2692";
      LAR2  LD 1;
      L     DIW [AR2,P#2050.0];
      OPN   DI 2292;
      T     DIW 6;
      OPN   DI [LW 5];
      L     DID [AR2,P#2052.0];
      OPN   DI 6004;
      T     DID 560;
      OPN   DI [LW 5];
      L     DIW [AR2,P#2056.0];
      OPN   DI 6004;
      T     DIW 564;
      OPN   DI [LW 5];
      A     DIX [AR2,P#2060.0];
      OPN   DI 7006;
      =     DIX 5.3;
      OPN   DI [LW 5];
      A     DIX [AR2,P#2060.1];
      OPN   DI 2555;
      =     DIX 3.5;
      OPN   DI [LW 5];
      CDB;
      BLD   15;
      NOP   0;
NETWORK
TITLE = T6_XPF_A1
      A     "Always0";
      =     L 0.0;
      BLD   103;
      A     "IMCC_LOCK".T6_D_A2_Open;
      =     L 0.1;
      BLD   103;
      A     "Maste_To_Slave_Mod_DB".FireAlarm;
      =     L 0.2;
      BLD   103;
      A     "Maste_To_Slave_Mod_DB".BlockAlarm;
      =     L 0.3;
      BLD   103;
      BLD   14;
      =     L 7.0;
      L     DINO;
      T     LW 5;
      CDB;
      OPN   DI [LW 5];
      TAR2  LD 1;
      A     L 0.0;
      =     DIX [AR2,P#2146.0];
      BLD   11;
      L     W#16#1002;
      T     LW 10;
      L     8;
      T     LW 12;
      L     2291;
      T     LW 14;
      L     P#DBX 52.0;
      T     LD 16;
      L     W#16#1002;
      T     LW 20;
      L     8;
      T     LW 22;
      L     DINO;
      T     LW 24;
      +AR2  P#2148.0;
      TAR2;
      LAR2  LD 1;
      T     LD 26;
      UC    "BLKMOV";
      {     P#L 10.0, P#L 8.0, P#L 20.0 };
      L     580;
      T     DIW [AR2,P#2156.0];
      OPN   DI 6040;
      L     DIW 230;
      OPN   DI [LW 5];
      T     DIW [AR2,P#2158.0];
      BLD   11;
      L     W#16#1002;
      T     LW 10;
      L     2;
      T     LW 12;
      L     7004;
      T     LW 14;
      L     P#DBX 64.0;
      T     LD 16;
      L     W#16#1002;
      T     LW 20;
      L     2;
      T     LW 22;
      L     DINO;
      T     LW 24;
      +AR2  P#2160.0;
      TAR2;
      LAR2  LD 1;
      T     LD 26;
      UC    "BLKMOV";
      {     P#L 10.0, P#L 8.0, P#L 20.0 };
      BLD   11;
      L     W#16#1002;
      T     LW 10;
      L     2;
      T     LW 12;
      L     7005;
      T     LW 14;
      L     P#DBX 6.0;
      T     LD 16;
      L     W#16#1002;
      T     LW 20;
      L     2;
      T     LW 22;
      L     DINO;
      T     LW 24;
      +AR2  P#2162.0;
      TAR2;
      LAR2  LD 1;
      T     LD 26;
      UC    "BLKMOV";
      {     P#L 10.0, P#L 8.0, P#L 20.0 };
      A     L 0.1;
      =     DIX [AR2,P#2164.0];
      L     DBD [AR2,P#0.0];
      T     DID [AR2,P#2166.0];
      BLD   11;
      L     W#16#1002;
      T     LW 10;
      L     2;
      T     LW 12;
      L     7005;
      T     LW 14;
      L     P#DBX 36.0;
      T     LD 16;
      L     W#16#1002;
      T     LW 20;
      L     2;
      T     LW 22;
      L     DINO;
      T     LW 24;
      +AR2  P#2170.0;
      TAR2;
      LAR2  LD 1;
      T     LD 26;
      UC    "BLKMOV";
      {     P#L 10.0, P#L 8.0, P#L 20.0 };
      OPN   DI 7005;
      L     DIW 312;
      OPN   DI [LW 5];
      T     DIW [AR2,P#2172.0];
      A     L 0.2;
      =     DIX [AR2,P#2174.0];
      A     L 0.3;
      =     DIX [AR2,P#2174.1];
      +AR2  P#2146.0;
      UC    "HF3_IMCC_FJ_FB2692";
      LAR2  LD 1;
      L     DIW [AR2,P#2176.0];
      OPN   DI 2292;
      T     DIW 16;
      OPN   DI [LW 5];
      L     DID [AR2,P#2178.0];
      OPN   DI 6004;
      T     DID 588;
      OPN   DI [LW 5];
      L     DIW [AR2,P#2182.0];
      OPN   DI 6004;
      T     DIW 592;
      OPN   DI [LW 5];
      A     DIX [AR2,P#2186.0];
      OPN   DI 7006;
      =     DIX 5.4;
      OPN   DI [LW 5];
      A     DIX [AR2,P#2186.1];
      OPN   DI 2555;
      =     DIX 3.4;
      OPN   DI [LW 5];
      CDB;
      BLD   15;
      NOP   0;
NETWORK
TITLE = T7_SPF_A1
      A     "Always0";
      =     L 0.0;
      BLD   103;
      A     "IMCC_LOCK".T7_D_A1_Open;
      =     L 0.1;
      BLD   103;
      A     "Maste_To_Slave_Mod_DB".FireAlarm;
      =     L 0.2;
      BLD   103;
      A     "Maste_To_Slave_Mod_DB".BlockAlarm;
      =     L 0.3;
      BLD   103;
      BLD   14;
      =     L 7.0;
      L     DINO;
      T     LW 5;
      CDB;
      OPN   DI [LW 5];
      TAR2  LD 1;
      A     L 0.0;
      =     DIX [AR2,P#2272.0];
      BLD   11;
      L     W#16#1002;
      T     LW 10;
      L     8;
      T     LW 12;
      L     2291;
      T     LW 14;
      L     P#DBX 60.0;
      T     LD 16;
      L     W#16#1002;
      T     LW 20;
      L     8;
      T     LW 22;
      L     DINO;
      T     LW 24;
      +AR2  P#2274.0;
      TAR2;
      LAR2  LD 1;
      T     LD 26;
      UC    "BLKMOV";
      {     P#L 10.0, P#L 8.0, P#L 20.0 };
      L     594;
      T     DIW [AR2,P#2282.0];
      OPN   DI 6040;
      L     DIW 238;
      OPN   DI [LW 5];
      T     DIW [AR2,P#2284.0];
      BLD   11;
      L     W#16#1002;
      T     LW 10;
      L     2;
      T     LW 12;
      L     7004;
      T     LW 14;
      L     P#DBX 72.0;
      T     LD 16;
      L     W#16#1002;
      T     LW 20;
      L     2;
      T     LW 22;
      L     DINO;
      T     LW 24;
      +AR2  P#2286.0;
      TAR2;
      LAR2  LD 1;
      T     LD 26;
      UC    "BLKMOV";
      {     P#L 10.0, P#L 8.0, P#L 20.0 };
      BLD   11;
      L     W#16#1002;
      T     LW 10;
      L     2;
      T     LW 12;
      L     7005;
      T     LW 14;
      L     P#DBX 8.0;
      T     LD 16;
      L     W#16#1002;
      T     LW 20;
      L     2;
      T     LW 22;
      L     DINO;
      T     LW 24;
      +AR2  P#2288.0;
      TAR2;
      LAR2  LD 1;
      T     LD 26;
      UC    "BLKMOV";
      {     P#L 10.0, P#L 8.0, P#L 20.0 };
      A     L 0.1;
      =     DIX [AR2,P#2290.0];
      L     DBD [AR2,P#0.0];
      T     DID [AR2,P#2292.0];
      BLD   11;
      L     W#16#1002;
      T     LW 10;
      L     2;
      T     LW 12;
      L     7005;
      T     LW 14;
      L     P#DBX 38.0;
      T     LD 16;
      L     W#16#1002;
      T     LW 20;
      L     2;
      T     LW 22;
      L     DINO;
      T     LW 24;
      +AR2  P#2296.0;
      TAR2;
      LAR2  LD 1;
      T     LD 26;
      UC    "BLKMOV";
      {     P#L 10.0, P#L 8.0, P#L 20.0 };
      OPN   DI 7005;
      L     DIW 312;
      OPN   DI [LW 5];
      T     DIW [AR2,P#2298.0];
      A     L 0.2;
      =     DIX [AR2,P#2300.0];
      A     L 0.3;
      =     DIX [AR2,P#2300.1];
      +AR2  P#2272.0;
      UC    "HF3_IMCC_FJ_FB2692";
      LAR2  LD 1;
      L     DIW [AR2,P#2302.0];
      OPN   DI 2292;
      T     DIW 18;
      OPN   DI [LW 5];
      L     DID [AR2,P#2304.0];
      OPN   DI 6004;
      T     DID 602;
      OPN   DI [LW 5];
      L     DIW [AR2,P#2308.0];
      OPN   DI 6004;
      T     DIW 606;
      OPN   DI [LW 5];
      A     DIX [AR2,P#2312.0];
      OPN   DI 7006;
      =     DIX 5.7;
      OPN   DI [LW 5];
      A     DIX [AR2,P#2312.1];
      OPN   DI 2555;
      =     DIX 4.0;
      OPN   DI [LW 5];
      CDB;
      BLD   15;
      NOP   0;
END_FUNCTION_BLOCK

FUNCTION_BLOCK "HF3_IMCC_FJ_FB2692"	// FB 2692
VERSION : 0.1
VAR_INPUT
  Main : BOOL ;	//1为大端  0为小端
  IN_RD : ARRAY  [0 .. 3 ] OF WORD ;
  HMI_Adr : INT ;
  SCtrl : WORD ;
  MCtrl : ARRAY  [0 .. 3 ] OF //0-模式启动1-模式停止
  BOOL ;
  Mode : ARRAY  [0 .. 15 ] OF //0-模式开始1-模式结束2-模式执行中
  BOOL ;
  Open : BOOL ;	//连锁风阀开/设定位
  PT : TIME ;	//设备动作超时时间
  ALL : ARRAY  [0 .. 15 ] OF //0-一键单控1-一键模控2-时间表控制
  BOOL ;
  H_P_All_Ctrl : WORD ;	//全局命令
  FireAlarm : BOOL ;	//火灾信号
  BlockAlarm : BOOL ;	//阻塞信号
END_VAR
VAR_OUTPUT
  qnWR : WORD ;	//控制输出命令
  RT : REAL ;	//设备运行时间
  SumFlt : INT ;	//故障次数
  SumRun : INT ;	//启动次数
  Refuse : BOOL ;	//模式不符
  stop : BOOL ;
END_VAR
VAR
  IN_RD1 : WORD ;
  qtWR : WORD ;
  TOHMI : WORD ;
  qtwr_temp : WORD ;
  SFlag : BOOL ;	//单控标志
  SingTout : BOOL ;	//单控超时
  Timeout : BOOL ;	//设备动作超时
  DI_Temp : ARRAY  [0 .. 15 ] OF //设备动作字
  BOOL ;
  DO_Temp : ARRAY  [0 .. 15 ] OF //1-启动控制2-停止控制
  BOOL ;
  Ctrl : ARRAY  [0 .. 15 ] OF //0-启动命令1-停止命令
  BOOL ;
  SCtrl_Temp : ARRAY  [0 .. 15 ] OF //上位命令解析
  BOOL ;
  Latch : ARRAY  [0 .. 7 ] OF //0-单控启动锁定1-单控停止锁定
  BOOL ;
  McFlag : BOOL ;	//检修牌
  QTout : BOOL ;	//输出超时
  H_P_All_Ctrl_Temp : ARRAY  [0 .. 15 ] OF BOOL ;
  Ton1 : SFB 4;
  Ton2 : SFB 4;
  RunFaultSum : FB 2006;
END_VAR
VAR_TEMP
  AR2_Value : DWORD ;
  DI_NO : INT ;
  Data_Len : INT ;
  DB_NO : INT ;
END_VAR
BEGIN
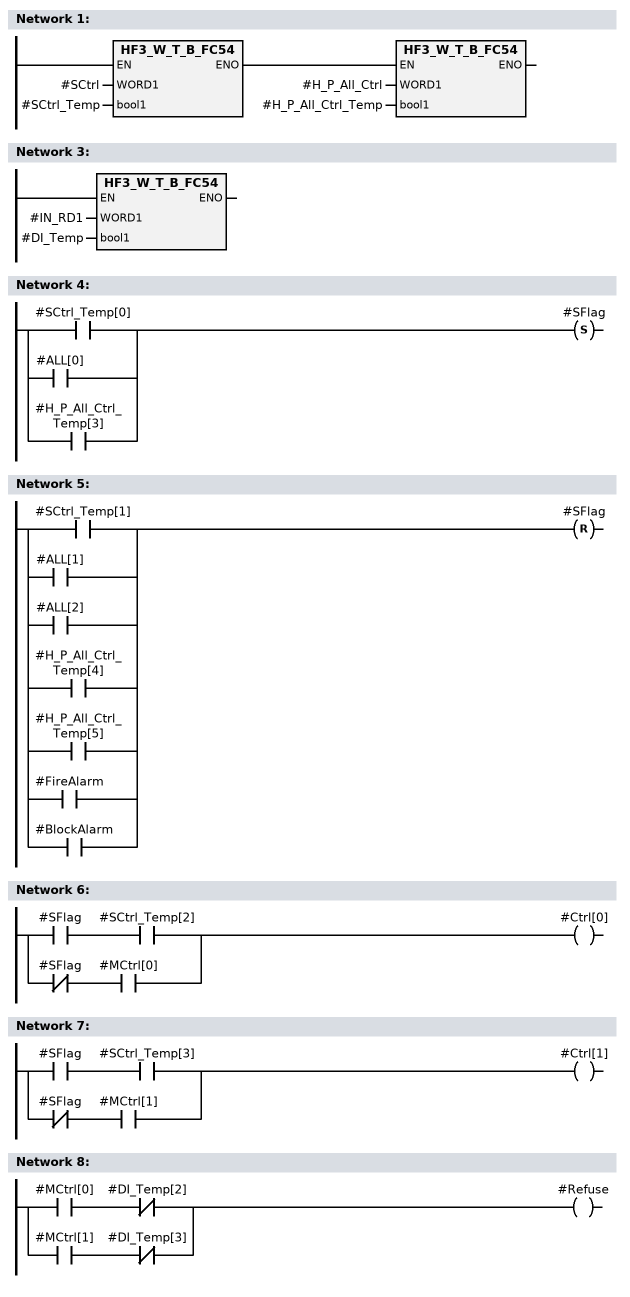
NETWORK
TITLE =
      A(;
      CALL  "HF3_W_T_B_FC54" (
           WORD1                    := #SCtrl,
           bool1                    := #SCtrl_Temp);
      A     BR;
      );
      JNB   _001;
      CALL  "HF3_W_T_B_FC54" (
           WORD1                    := #H_P_All_Ctrl,
           bool1                    := #H_P_All_Ctrl_Temp);
_001: NOP   0;
NETWORK
TITLE =
//第1个字BIT 0BAS远程
//第1个字BIT 1就地模式
//第1个字BIT 2运行状态
//第1个字BIT 3停车状态
//第1个字BIT 4故障
//
//
//第2个字电机A相电流（A）
//第3个字电机B相电流（A）
//第4个字电机C相电流（A）
//
      TAR2;
      T     #AR2_Value;
      L     6002;
      T     #DB_NO;
      A     #Main;	//此端是否为大端
      JC    big;
      L     6004;
      T     #DB_NO;
big:  L     DINO;	//存储背景数据块号
      T     #DI_NO;
      OPN   DB [#DB_NO];	//打开
      L     #HMI_Adr;
      SLD   3;
      LAR1;
// *********************小风机中DI状态读取**********************
      L     #IN_RD[0];	//第一个字中包含数字量信息
      T     #IN_RD1;
//初始化AR2寄存器用于AI量传递
      TAR2;
      AD    DW#16#FFFFFF;
      L     P##IN_RD;
      +D;
      OD    DW#16#85000000;
      LAR2;
//*********************小风机中AI状态读取**********************
//读取模拟量输入
      L     3;
ilop: T     #Data_Len;
      L     W [AR2,P#2.0];	//智能低压点表新更新，第二个字开始为模拟量
      T     DBW [AR1,P#2.0];
      +AR1  P#2.0;
      +AR2  P#2.0;
      L     #Data_Len;
      LOOP  ilop;
//恢复AR2 DI寄存器
      L     #AR2_Value;
      LAR2;
//     OPN   DI [#DI_NO]
NETWORK
TITLE =
      CALL  "HF3_W_T_B_FC54" (
           WORD1                    := #IN_RD1,
           bool1                    := #DI_Temp);
      NOP   0;
NETWORK
TITLE =
      O     #SCtrl_Temp[0];
      O     #ALL[0];
      O     #H_P_All_Ctrl_Temp[3];
      S     #SFlag;
NETWORK
TITLE =
      O     #SCtrl_Temp[1];
      O     #ALL[1];
      O     #ALL[2];
      O     #H_P_All_Ctrl_Temp[4];
      O     #H_P_All_Ctrl_Temp[5];
      O     #FireAlarm;
      O     #BlockAlarm;
      R     #SFlag;
NETWORK
TITLE =
      A     #SFlag;
      A     #SCtrl_Temp[2];
      O;
      AN    #SFlag;
      A     #MCtrl[0];
      =     #Ctrl[0];
NETWORK
TITLE =
      A     #SFlag;
      A     #SCtrl_Temp[3];
      O;
      AN    #SFlag;
      A     #MCtrl[1];
      =     #Ctrl[1];
NETWORK
TITLE =
      A     #MCtrl[0];
      AN    #DI_Temp[2];
      O;
      A     #MCtrl[1];
      AN    #DI_Temp[3];
      =     #Refuse;
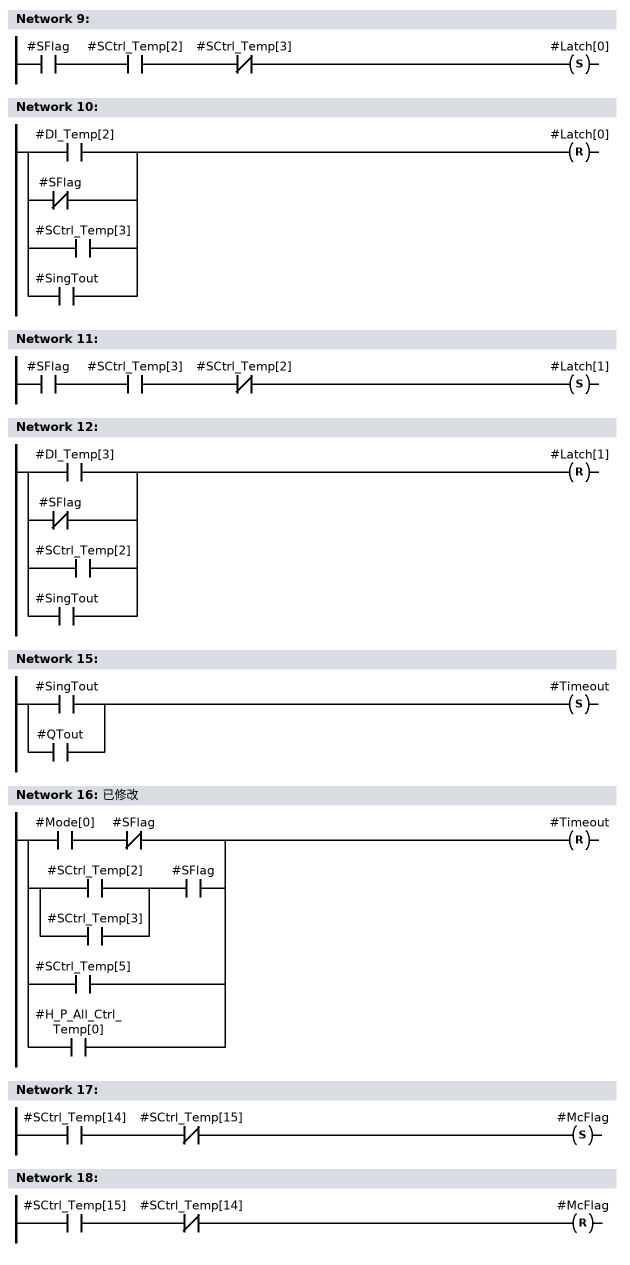
NETWORK
TITLE =
      A     #SFlag;
      A     #SCtrl_Temp[2];
      AN    #SCtrl_Temp[3];
      S     #Latch[0];
NETWORK
TITLE =
      O     #DI_Temp[2];
      ON    #SFlag;
      O     #SCtrl_Temp[3];
      O     #SingTout;
      R     #Latch[0];
NETWORK
TITLE =
      A     #SFlag;
      A     #SCtrl_Temp[3];
      AN    #SCtrl_Temp[2];
      S     #Latch[1];
NETWORK
TITLE =
      O     #DI_Temp[3];
      ON    #SFlag;
      O     #SCtrl_Temp[2];
      O     #SingTout;
      R     #Latch[1];
NETWORK
TITLE =
      A(;
      O     #Latch[0];
      O     #Latch[1];
      );
      =     L 10.0;
      BLD   103;
      BLD   16;
      =     L 17.0;
      L     DINO;
      T     LW 15;
      CDB;
      OPN   DI [LW 15];
      TAR2  LD 11;
      A     L 10.0;
      =     DIX [AR2,P#66.0];
      L     DBD [AR2,P#20.0];
      T     DID [AR2,P#68.0];
      +AR2  P#66.0;
      UC    "TON";
      LAR2  LD 11;
      A     DIX [AR2,P#72.0];
      =     DBX [AR2,P#50.1];
      CDB;
      BLD   17;
      NOP   0;
NETWORK
TITLE =
      A(;
      O     #DO_Temp[0];
      O     #DO_Temp[1];
      );
      =     L 10.0;
      BLD   103;
      BLD   16;
      =     L 17.0;
      L     DINO;
      T     LW 15;
      CDB;
      OPN   DI [LW 15];
      TAR2  LD 11;
      A     L 10.0;
      =     DIX [AR2,P#88.0];
      L     DBD [AR2,P#20.0];
      T     DID [AR2,P#90.0];
      +AR2  P#88.0;
      UC    "TON";
      LAR2  LD 11;
      A     DIX [AR2,P#94.0];
      =     DBX [AR2,P#62.1];
      CDB;
      BLD   17;
      NOP   0;
NETWORK
TITLE =
      O     #SingTout;
      O     #QTout;
      S     #Timeout;
NETWORK
TITLE = 已修改
      A     #Mode[0];
      AN    #SFlag;
      O;
      A(;
      O     #SCtrl_Temp[2];
      O     #SCtrl_Temp[3];
      );
      A     #SFlag;
      O     #SCtrl_Temp[5];
      O     #H_P_All_Ctrl_Temp[0];
      R     #Timeout;
NETWORK
TITLE =
      A     #SCtrl_Temp[14];
      AN    #SCtrl_Temp[15];
      S     #McFlag;
NETWORK
TITLE =
      A     #SCtrl_Temp[15];
      AN    #SCtrl_Temp[14];
      R     #McFlag;
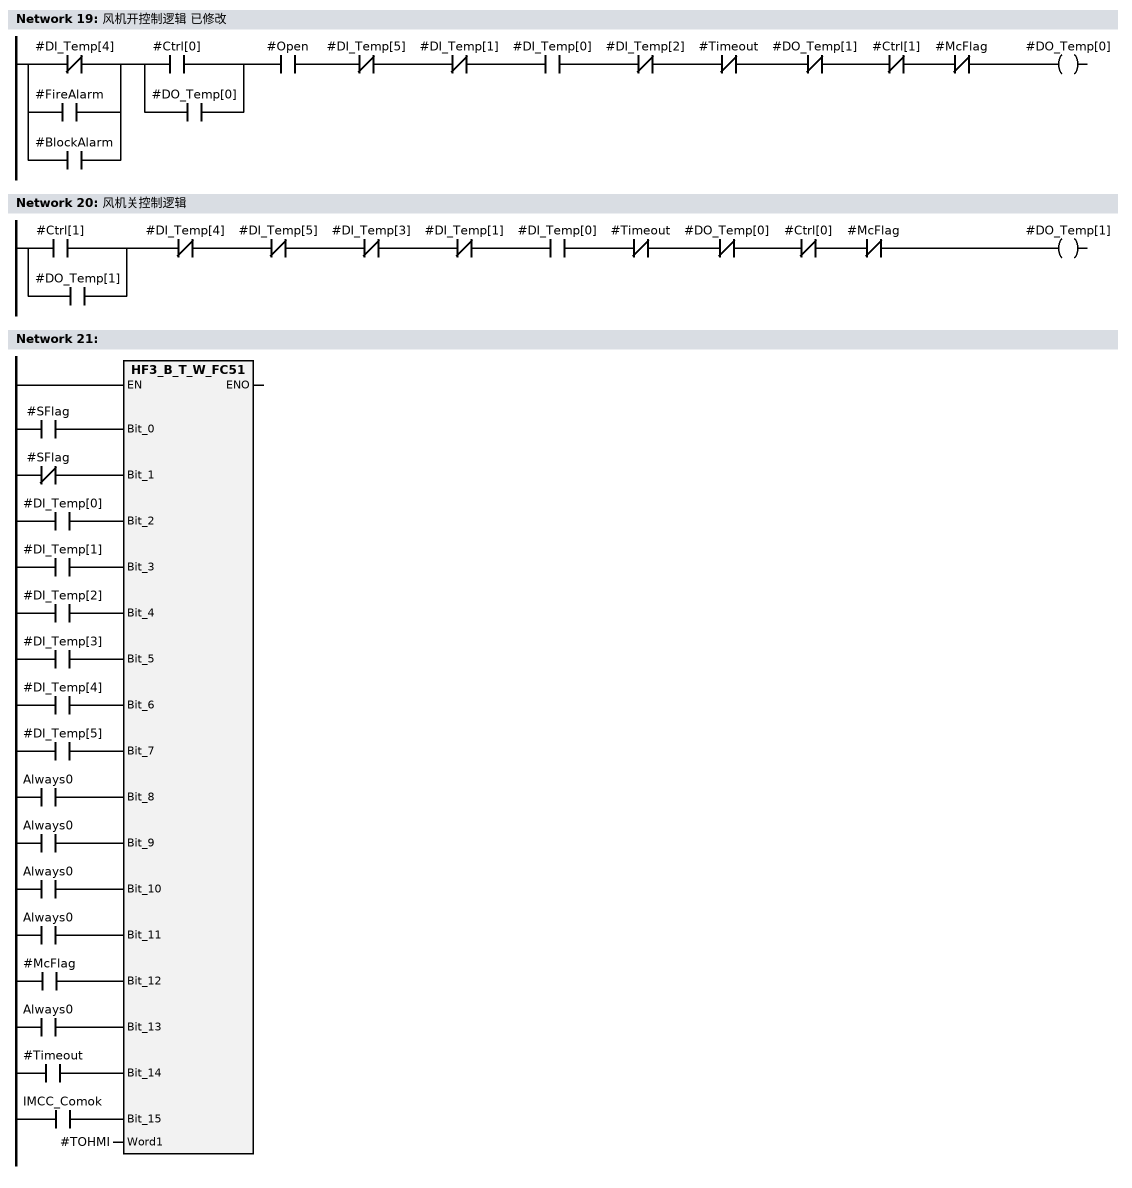
NETWORK
TITLE = 风机开控制逻辑 已修改
      A(;
      ON    #DI_Temp[4];
      O     #FireAlarm;
      O     #BlockAlarm;
      );
      A(;
      O     #Ctrl[0];
      O     #DO_Temp[0];
      );
      A     #Open;
      AN    #DI_Temp[5];
      AN    #DI_Temp[1];
      A     #DI_Temp[0];
      AN    #DI_Temp[2];
      AN    #Timeout;
      AN    #DO_Temp[1];
      AN    #Ctrl[1];
      AN    #McFlag;
      =     #DO_Temp[0];
NETWORK
TITLE = 风机关控制逻辑
      A(;
      O     #Ctrl[1];
      O     #DO_Temp[1];
      );
      AN    #DI_Temp[4];
      AN    #DI_Temp[5];
      AN    #DI_Temp[3];
      AN    #DI_Temp[1];
      A     #DI_Temp[0];
      AN    #Timeout;
      AN    #DO_Temp[0];
      AN    #Ctrl[0];
      AN    #McFlag;
      =     #DO_Temp[1];
NETWORK
TITLE =
      A     #SFlag;
      =     L 10.0;
      BLD   103;
      AN    #SFlag;
      =     L 10.1;
      BLD   103;
      A     #DI_Temp[0];
      =     L 10.2;
      BLD   103;
      A     #DI_Temp[1];
      =     L 10.3;
      BLD   103;
      A     #DI_Temp[2];
      =     L 10.4;
      BLD   103;
      A     #DI_Temp[3];
      =     L 10.5;
      BLD   103;
      A     #DI_Temp[4];
      =     L 10.6;
      BLD   103;
      A     #DI_Temp[5];
      =     L 10.7;
      BLD   103;
      A     "Always0";
      =     L 11.0;
      BLD   103;
      A     "Always0";
      =     L 11.1;
      BLD   103;
      A     "Always0";
      =     L 11.2;
      BLD   103;
      A     "Always0";
      =     L 11.3;
      BLD   103;
      A     #McFlag;
      =     L 11.4;
      BLD   103;
      A     "Always0";
      =     L 11.5;
      BLD   103;
      A     #Timeout;
      =     L 11.6;
      BLD   103;
      A     "IMCC_Comok";
      =     L 11.7;
      BLD   103;
      CALL  "HF3_B_T_W_FC51" (
           Bit_0                    := L 10.0,
           Bit_1                    := L 10.1,
           Bit_2                    := L 10.2,
           Bit_3                    := L 10.3,
           Bit_4                    := L 10.4,
           Bit_5                    := L 10.5,
           Bit_6                    := L 10.6,
           Bit_7                    := L 10.7,
           Bit_8                    := L 11.0,
           Bit_9                    := L 11.1,
           Bit_10                   := L 11.2,
           Bit_11                   := L 11.3,
           Bit_12                   := L 11.4,
           Bit_13                   := L 11.5,
           Bit_14                   := L 11.6,
           Bit_15                   := L 11.7,
           Word1                    := #TOHMI);
      NOP   0;
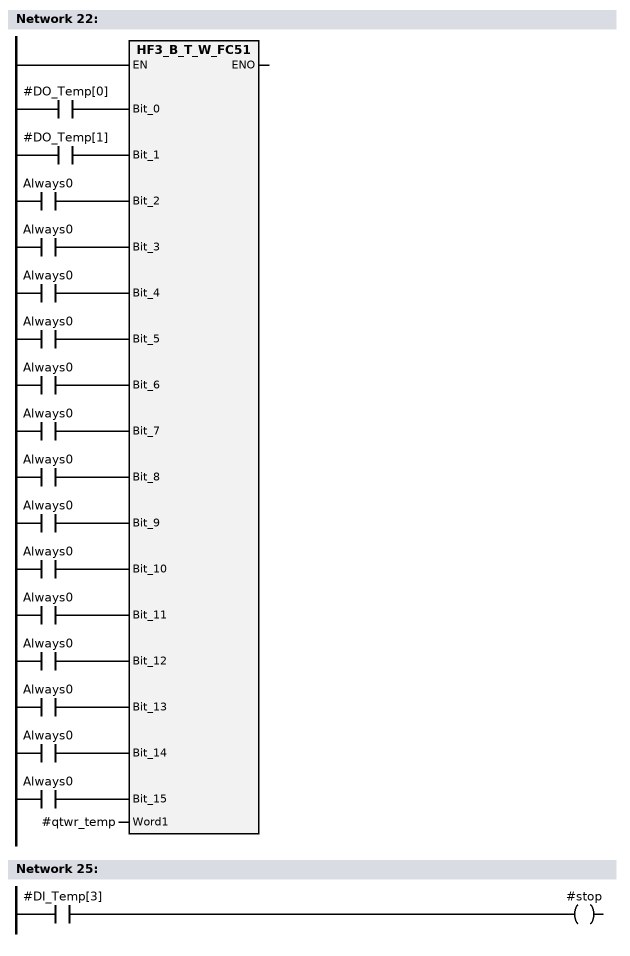
NETWORK
TITLE =
      A     #DO_Temp[0];
      =     L 10.0;
      BLD   103;
      A     #DO_Temp[1];
      =     L 10.1;
      BLD   103;
      A     "Always0";
      =     L 10.2;
      BLD   103;
      A     "Always0";
      =     L 10.3;
      BLD   103;
      A     "Always0";
      =     L 10.4;
      BLD   103;
      A     "Always0";
      =     L 10.5;
      BLD   103;
      A     "Always0";
      =     L 10.6;
      BLD   103;
      A     "Always0";
      =     L 10.7;
      BLD   103;
      A     "Always0";
      =     L 11.0;
      BLD   103;
      A     "Always0";
      =     L 11.1;
      BLD   103;
      A     "Always0";
      =     L 11.2;
      BLD   103;
      A     "Always0";
      =     L 11.3;
      BLD   103;
      A     "Always0";
      =     L 11.4;
      BLD   103;
      A     "Always0";
      =     L 11.5;
      BLD   103;
      A     "Always0";
      =     L 11.6;
      BLD   103;
      A     "Always0";
      =     L 11.7;
      BLD   103;
      CALL  "HF3_B_T_W_FC51" (
           Bit_0                    := L 10.0,
           Bit_1                    := L 10.1,
           Bit_2                    := L 10.2,
           Bit_3                    := L 10.3,
           Bit_4                    := L 10.4,
           Bit_5                    := L 10.5,
           Bit_6                    := L 10.6,
           Bit_7                    := L 10.7,
           Bit_8                    := L 11.0,
           Bit_9                    := L 11.1,
           Bit_10                   := L 11.2,
           Bit_11                   := L 11.3,
           Bit_12                   := L 11.4,
           Bit_13                   := L 11.5,
           Bit_14                   := L 11.6,
           Bit_15                   := L 11.7,
           Word1                    := #qtwr_temp);
      NOP   0;
NETWORK
TITLE =
//控制命令输出
      CLR;
      L     #SCtrl;
      L     W#16#ABCD;
      <>I;
      JC    seiz;
      L     W#16#0;
      T     #qtwr_temp;
seiz: L     #qtwr_temp;
      T     #qnWR;
//tohmi输出
      L     #HMI_Adr;
      SLD   3;
      LAR1;
      OPN   DB [#DB_NO];
      L     #TOHMI;
      T     DBW [AR1,P#0.0];
NETWORK
TITLE =
      A     #DI_Temp[2];
      =     L 10.0;
      BLD   103;
      A     #DI_Temp[4];
      =     L 10.1;
      BLD   103;
      A     M 20.5;
      =     L 10.2;
      BLD   103;
      A     #SCtrl_Temp[12];
      =     L 10.4;
      BLD   103;
      A     #SCtrl_Temp[13];
      =     L 10.5;
      BLD   103;
      BLD   14;
      =     L 17.0;
      L     DINO;
      T     LW 15;
      CDB;
      OPN   DI [LW 15];
      TAR2  LD 11;
      A     L 10.0;
      =     DIX [AR2,P#110.0];
      A     L 10.1;
      =     DIX [AR2,P#110.1];
      A     L 10.2;
      =     DIX [AR2,P#110.2];
      A     L 10.4;
      =     DIX [AR2,P#110.4];
      A     L 10.5;
      =     DIX [AR2,P#110.5];
      +AR2  P#110.0;
      UC    "HF3_RunFaultSum";
      LAR2  LD 11;
      L     DID [AR2,P#112.0];
      T     DBD [AR2,P#32.0];
      L     DIW [AR2,P#116.0];
      T     DBW [AR2,P#38.0];
      L     DIW [AR2,P#118.0];
      T     DBW [AR2,P#36.0];
      CDB;
      BLD   15;
      NOP   0;
NETWORK
TITLE =
      A     #DI_Temp[3];
      =     #stop;
END_FUNCTION_BLOCK

FUNCTION_BLOCK "HF3_IMCC_DZ_FB2701"	// FB 2701
TITLE = IMCC系统电动组合风阀
VERSION : 0.1
VAR
  DZ_225_A1 : FB 2702;
  DZ_225_A2 : FB 2702;
  DZ_225_A3 : FB 2702;
  DZ_225_A4 : FB 2702;
  DZ_225_A5 : FB 2702;
  DZ_225_A6 : FB 2702;
  DZ_225_A7 : FB 2702;
  DZ_225_A8 : FB 2702;
  PT : TIME  := T#45S;
END_VAR
BEGIN
NETWORK
TITLE =
NETWORK
TITLE =
NETWORK
TITLE =
NETWORK
TITLE =
NETWORK
TITLE =
NETWORK
TITLE =
NETWORK
TITLE =
NETWORK
TITLE =
END_FUNCTION_BLOCK

FUNCTION_BLOCK "HF3_IMCC_DZ_B2702"	// FB 2702
VERSION : 0.1
VAR_INPUT
  SCtrl : WORD ;	//控制命令
  inRD : WORD ;	//风阀反馈信息
  H_P_ALL_Ctrl : WORD ;	//全局命令
  Stop : BOOL ;	//连锁信号
  FireAlarm : BOOL ;	//火灾信号
  BlockAlarm : BOOL ;	//阻塞信号
  MCtrl : ARRAY  [0 .. 3 ] OF //0-开阀1-关阀
  BOOL ;
  Mode : ARRAY  [0 .. 15 ] OF //0-开始1-结束2-执行中
  BOOL ;
  ALL : ARRAY  [0 .. 15 ] OF //单系统命令
  BOOL ;
  PT : TIME ;	//设备动作超时
  commok : BOOL ;
END_VAR
VAR_OUTPUT
  qtWR : WORD ;	//阀控制信息
  ToHMI : WORD ;	//给上位信号
  Refuse : BOOL ;	//模式不符
  Open : BOOL ;	//阀控制信息
END_VAR
VAR
  SCtrl_Temp : ARRAY  [0 .. 15 ] OF //01-单模23-开关
  BOOL ;
  DI_Temp : ARRAY  [0 .. 15 ] OF //23-开关
  BOOL ;
  DO_Temp : ARRAY  [0 .. 15 ] OF //1-开2-关输出
  BOOL ;
  H_P_ALL_Ctrl_Temp : ARRAY  [0 .. 15 ] OF BOOL ;
  Ctrl : ARRAY  [0 .. 15 ] OF //开关控制
  BOOL ;
  Latch : ARRAY  [0 .. 15 ] OF //控制锁定
  BOOL ;
  Ton2 : SFB 4;
  TON1 : SFB 4;
  TON3 : SFB 4;
  TON4 : SFB 4;
  SFlag : BOOL ;	//单模控标志
  QTout : BOOL ;
  Timeout : BOOL ;	//设备动作超时
  McFlag : BOOL ;	//检修牌
  SIngTout : BOOL ;
END_VAR
BEGIN
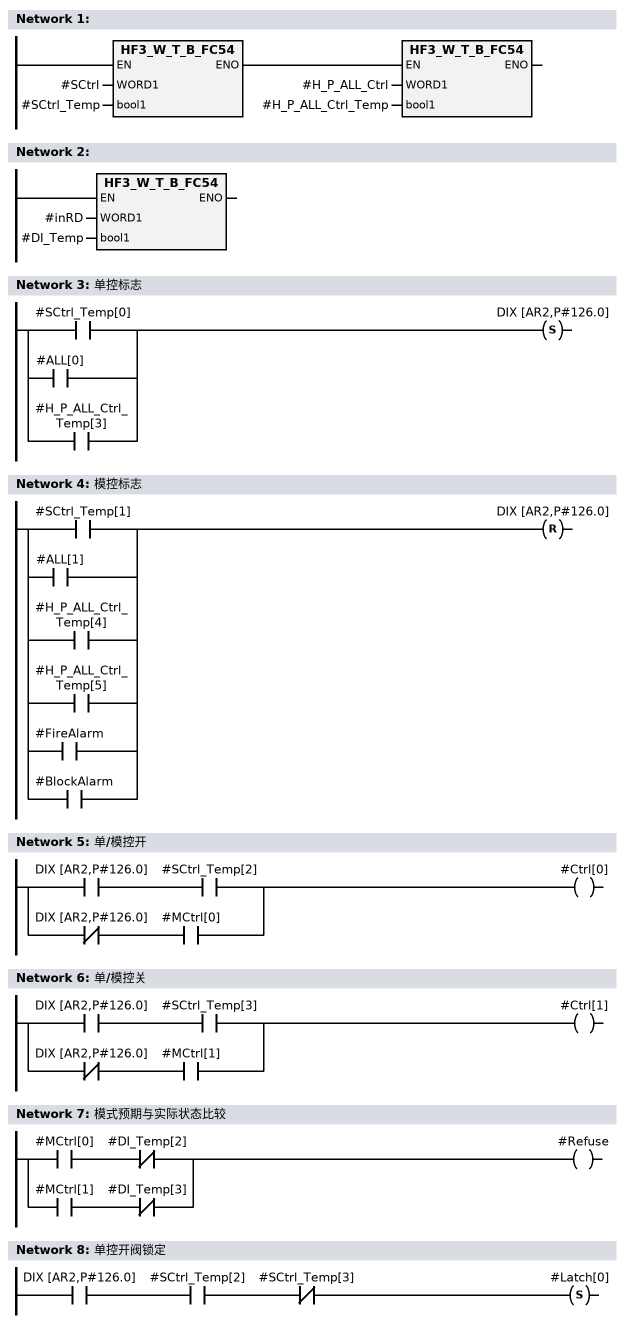
NETWORK
TITLE =
      A(;
      CALL  "HF3_W_T_B_FC54" (
           WORD1                    := #SCtrl,
           bool1                    := #SCtrl_Temp);
      A     BR;
      );
      JNB   _001;
      CALL  "HF3_W_T_B_FC54" (
           WORD1                    := #H_P_ALL_Ctrl,
           bool1                    := #H_P_ALL_Ctrl_Temp);
_001: NOP   0;
NETWORK
TITLE =
      CALL  "HF3_W_T_B_FC54" (
           WORD1                    := #inRD,
           bool1                    := #DI_Temp);
      NOP   0;
NETWORK
TITLE = 单控标志
      O     #SCtrl_Temp[0];
      O     #ALL[0];
      O     #H_P_ALL_Ctrl_Temp[3];
      S     DIX [AR2,P#126.0];
NETWORK
TITLE = 模控标志
      O     #SCtrl_Temp[1];
      O     #ALL[1];
      O     #H_P_ALL_Ctrl_Temp[4];
      O     #H_P_ALL_Ctrl_Temp[5];
      O     #FireAlarm;
      O     #BlockAlarm;
      R     DIX [AR2,P#126.0];
NETWORK
TITLE = 单/模控开
      A     DIX [AR2,P#126.0];
      A     #SCtrl_Temp[2];
      O;
      AN    DIX [AR2,P#126.0];
      A     #MCtrl[0];
      =     #Ctrl[0];
NETWORK
TITLE = 单/模控关
      A     DIX [AR2,P#126.0];
      A     #SCtrl_Temp[3];
      O;
      AN    DIX [AR2,P#126.0];
      A     #MCtrl[1];
      =     #Ctrl[1];
NETWORK
TITLE = 模式预期与实际状态比较
      A     #MCtrl[0];
      AN    #DI_Temp[2];
      O;
      A     #MCtrl[1];
      AN    #DI_Temp[3];
      =     #Refuse;
NETWORK
TITLE = 单控开阀锁定
      A     DIX [AR2,P#126.0];
      A     #SCtrl_Temp[2];
      AN    #SCtrl_Temp[3];
      S     #Latch[0];
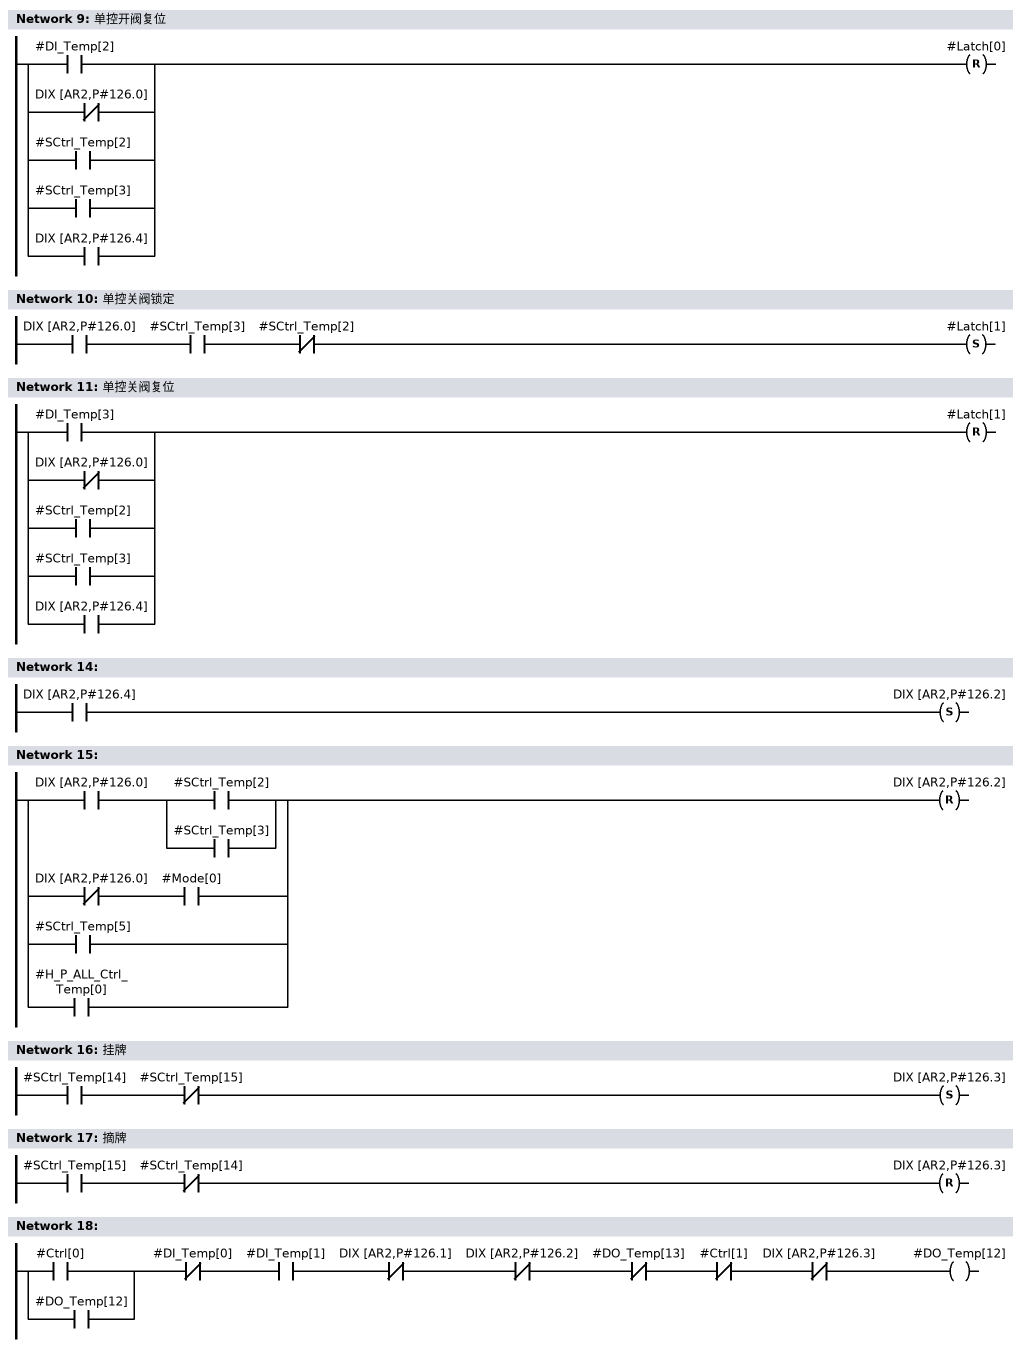
NETWORK
TITLE = 单控开阀复位
      O     #DI_Temp[2];
      ON    DIX [AR2,P#126.0];
      O     #SCtrl_Temp[2];
      O     #SCtrl_Temp[3];
      O     DIX [AR2,P#126.4];
      R     #Latch[0];
NETWORK
TITLE = 单控关阀锁定
      A     DIX [AR2,P#126.0];
      A     #SCtrl_Temp[3];
      AN    #SCtrl_Temp[2];
      S     #Latch[1];
NETWORK
TITLE = 单控关阀复位
      O     #DI_Temp[3];
      ON    DIX [AR2,P#126.0];
      O     #SCtrl_Temp[2];
      O     #SCtrl_Temp[3];
      O     DIX [AR2,P#126.4];
      R     #Latch[1];
NETWORK
TITLE =
      A(;
      O     #Latch[0];
      O     #Latch[1];
      );
      AN    #SCtrl_Temp[2];
      AN    #SCtrl_Temp[3];
      =     L 0.0;
      BLD   103;
      BLD   16;
      =     L 7.0;
      L     DINO;
      T     LW 5;
      CDB;
      OPN   DI [LW 5];
      TAR2  LD 1;
      A     L 0.0;
      =     DIX [AR2,P#60.0];
      L     L#90000;
      T     DID [AR2,P#62.0];
      +AR2  P#60.0;
      UC    "TON";
      LAR2  LD 1;
      A     DIX [AR2,P#66.0];
      =     DBX [AR2,P#126.4];
      CDB;
      BLD   17;
      NOP   0;
NETWORK
TITLE =
      A(;
      A     #DO_Temp[1];
      A     #DI_Temp[2];
      O;
      A     #DO_Temp[2];
      A     #DI_Temp[3];
      );
      =     L 0.0;
      BLD   103;
      BLD   16;
      =     L 7.0;
      L     DINO;
      T     LW 5;
      CDB;
      OPN   DI [LW 5];
      TAR2  LD 1;
      A     L 0.0;
      =     DIX [AR2,P#38.0];
      L     L#20000;
      T     DID [AR2,P#40.0];
      +AR2  P#38.0;
      UC    "TON";
      LAR2  LD 1;
      A     DIX [AR2,P#44.0];
      =     DBX [AR2,P#126.1];
      CDB;
      BLD   17;
      NOP   0;
NETWORK
TITLE =
      A     DIX [AR2,P#126.4];
      S     DIX [AR2,P#126.2];
NETWORK
TITLE =
      A     DIX [AR2,P#126.0];
      A(;
      O     #SCtrl_Temp[2];
      O     #SCtrl_Temp[3];
      );
      O;
      AN    DIX [AR2,P#126.0];
      A     #Mode[0];
      O     #SCtrl_Temp[5];
      O     #H_P_ALL_Ctrl_Temp[0];
      R     DIX [AR2,P#126.2];
NETWORK
TITLE = 挂牌
      A     #SCtrl_Temp[14];
      AN    #SCtrl_Temp[15];
      S     DIX [AR2,P#126.3];
NETWORK
TITLE = 摘牌
      A     #SCtrl_Temp[15];
      AN    #SCtrl_Temp[14];
      R     DIX [AR2,P#126.3];
NETWORK
TITLE =
      A(;
      O     #Ctrl[0];
      O     #DO_Temp[12];
      );
      AN    #DI_Temp[0];
      A     #DI_Temp[1];
      AN    DIX [AR2,P#126.1];
      AN    DIX [AR2,P#126.2];
      AN    #DO_Temp[13];
      AN    #Ctrl[1];
      AN    DIX [AR2,P#126.3];
      =     #DO_Temp[12];
NETWORK
TITLE =
      A     #DO_Temp[12];
      =     L 0.0;
      BLD   103;
      BLD   16;
      =     L 7.0;
      L     DINO;
      T     LW 5;
      CDB;
      OPN   DI [LW 5];
      TAR2  LD 1;
      A     L 0.0;
      =     DIX [AR2,P#82.0];
      L     L#1000;
      T     DID [AR2,P#84.0];
      +AR2  P#82.0;
      UC    "TON";
      LAR2  LD 1;
      A     DIX [AR2,P#88.0];
      =     DBX [AR2,P#30.1];
      CDB;
      BLD   17;
      NOP   0;
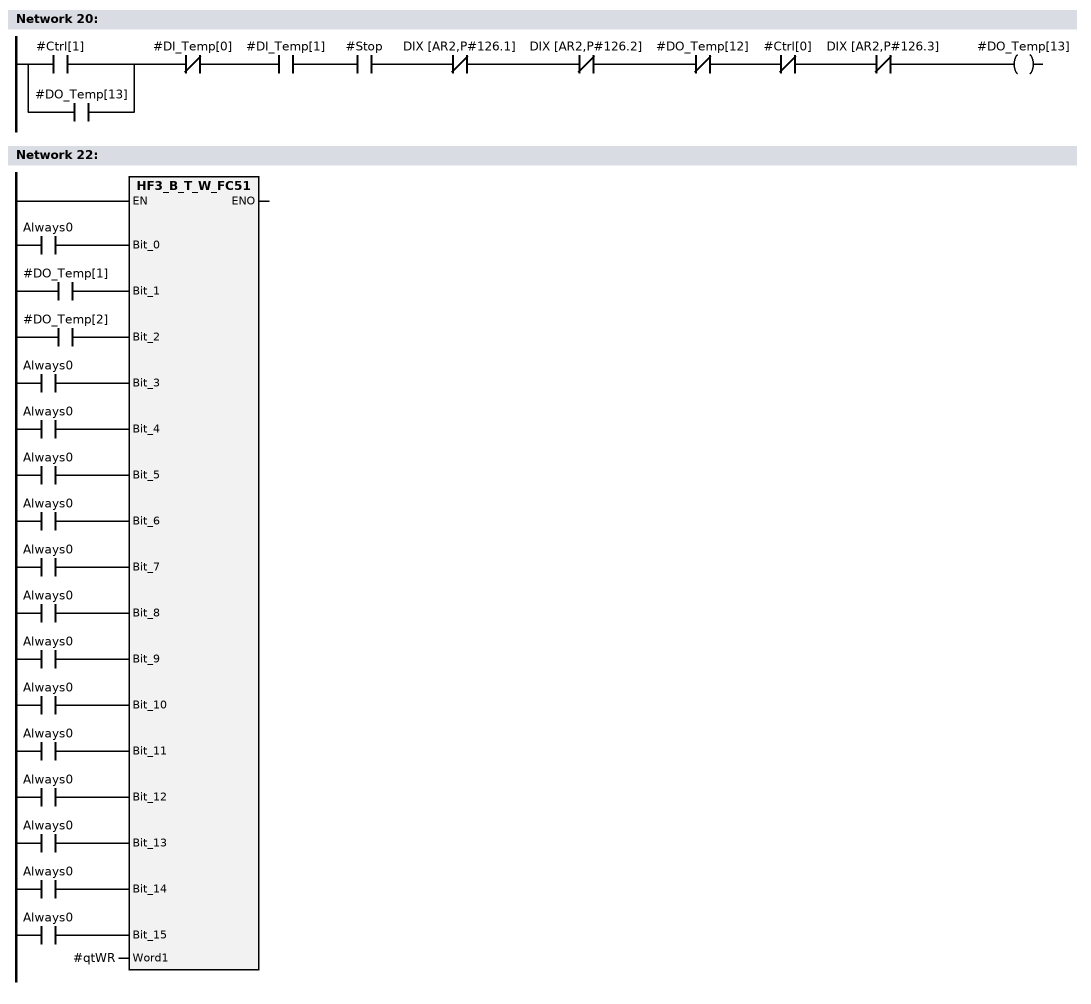
NETWORK
TITLE =
      A(;
      O     #Ctrl[1];
      O     #DO_Temp[13];
      );
      AN    #DI_Temp[0];
      A     #DI_Temp[1];
      A     #Stop;
      AN    DIX [AR2,P#126.1];
      AN    DIX [AR2,P#126.2];
      AN    #DO_Temp[12];
      AN    #Ctrl[0];
      AN    DIX [AR2,P#126.3];
      =     #DO_Temp[13];
NETWORK
TITLE =
      A     #DO_Temp[13];
      =     L 0.0;
      BLD   103;
      BLD   16;
      =     L 7.0;
      L     DINO;
      T     LW 5;
      CDB;
      OPN   DI [LW 5];
      TAR2  LD 1;
      A     L 0.0;
      =     DIX [AR2,P#104.0];
      L     L#1000;
      T     DID [AR2,P#106.0];
      +AR2  P#104.0;
      UC    "TON";
      LAR2  LD 1;
      A     DIX [AR2,P#110.0];
      =     DBX [AR2,P#30.2];
      CDB;
      BLD   17;
      NOP   0;
NETWORK
TITLE =
      A     "Always0";
      =     L 0.0;
      BLD   103;
      A     #DO_Temp[1];
      =     L 0.1;
      BLD   103;
      A     #DO_Temp[2];
      =     L 0.2;
      BLD   103;
      A     "Always0";
      =     L 0.3;
      BLD   103;
      A     "Always0";
      =     L 0.4;
      BLD   103;
      A     "Always0";
      =     L 0.5;
      BLD   103;
      A     "Always0";
      =     L 0.6;
      BLD   103;
      A     "Always0";
      =     L 0.7;
      BLD   103;
      A     "Always0";
      =     L 1.0;
      BLD   103;
      A     "Always0";
      =     L 1.1;
      BLD   103;
      A     "Always0";
      =     L 1.2;
      BLD   103;
      A     "Always0";
      =     L 1.3;
      BLD   103;
      A     "Always0";
      =     L 1.4;
      BLD   103;
      A     "Always0";
      =     L 1.5;
      BLD   103;
      A     "Always0";
      =     L 1.6;
      BLD   103;
      A     "Always0";
      =     L 1.7;
      BLD   103;
      CALL  "HF3_B_T_W_FC51" (
           Bit_0                    := L 0.0,
           Bit_1                    := L 0.1,
           Bit_2                    := L 0.2,
           Bit_3                    := L 0.3,
           Bit_4                    := L 0.4,
           Bit_5                    := L 0.5,
           Bit_6                    := L 0.6,
           Bit_7                    := L 0.7,
           Bit_8                    := L 1.0,
           Bit_9                    := L 1.1,
           Bit_10                   := L 1.2,
           Bit_11                   := L 1.3,
           Bit_12                   := L 1.4,
           Bit_13                   := L 1.5,
           Bit_14                   := L 1.6,
           Bit_15                   := L 1.7,
           Word1                    := #qtWR);
      NOP   0;
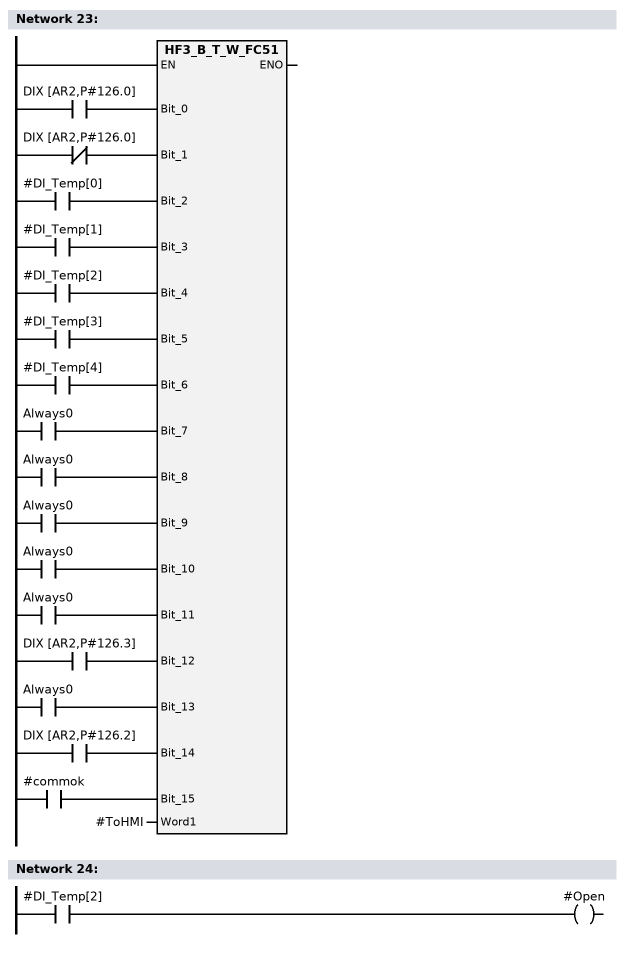
NETWORK
TITLE =
      A     DIX [AR2,P#126.0];
      =     L 0.0;
      BLD   103;
      AN    DIX [AR2,P#126.0];
      =     L 0.1;
      BLD   103;
      A     #DI_Temp[0];
      =     L 0.2;
      BLD   103;
      A     #DI_Temp[1];
      =     L 0.3;
      BLD   103;
      A     #DI_Temp[2];
      =     L 0.4;
      BLD   103;
      A     #DI_Temp[3];
      =     L 0.5;
      BLD   103;
      A     #DI_Temp[4];
      =     L 0.6;
      BLD   103;
      A     "Always0";
      =     L 0.7;
      BLD   103;
      A     "Always0";
      =     L 1.0;
      BLD   103;
      A     "Always0";
      =     L 1.1;
      BLD   103;
      A     "Always0";
      =     L 1.2;
      BLD   103;
      A     "Always0";
      =     L 1.3;
      BLD   103;
      A     DIX [AR2,P#126.3];
      =     L 1.4;
      BLD   103;
      A     "Always0";
      =     L 1.5;
      BLD   103;
      A     DIX [AR2,P#126.2];
      =     L 1.6;
      BLD   103;
      A     #commok;
      =     L 1.7;
      BLD   103;
      CALL  "HF3_B_T_W_FC51" (
           Bit_0                    := L 0.0,
           Bit_1                    := L 0.1,
           Bit_2                    := L 0.2,
           Bit_3                    := L 0.3,
           Bit_4                    := L 0.4,
           Bit_5                    := L 0.5,
           Bit_6                    := L 0.6,
           Bit_7                    := L 0.7,
           Bit_8                    := L 1.0,
           Bit_9                    := L 1.1,
           Bit_10                   := L 1.2,
           Bit_11                   := L 1.3,
           Bit_12                   := L 1.4,
           Bit_13                   := L 1.5,
           Bit_14                   := L 1.6,
           Bit_15                   := L 1.7,
           Word1                    := #ToHMI);
      NOP   0;
NETWORK
TITLE =
      A     #DI_Temp[2];
      =     #Open;
END_FUNCTION_BLOCK

